(* Logix 5000 project; controller TEC_81 vendor 1 type 14 code 148 rev 36.11; software revision 36.00 *)

TASK MainTask (continuous, watchdog 500 ms) : MainProgram, _05_Mesa_Central, _Almacen_2, _Almacen_1, Manu_camaras, CNC1_Prueba
TASK SafetyTask (periodic, rate 20 ms, priority 10, watchdog 20 ms) : SafetyProgram

MODULES
   Local : vendor 1 type 14 code 148 (ICP 1, rev 36.11)
      Ethernet : vendor 1 type 12 code 200 (ICP 0, Ethernet 10.12.143.10, rev 10.7, Input RPI 500 ms)
           Point_IO_Conveyor_2:4:I.0   // Cambio de Dirección Extendido Lado A Almacén
           Point_IO_Conveyor_2:4:I.1   // Cambio de Dirección Retraido Lado A Almacén
           Point_IO_Conveyor_2:4:I.2   // Sensor Inductivo Lado B CNC (Entrada)
           Point_IO_Conveyor_2:4:I.4   // Spare
           Point_IO_Conveyor_2:4:I.5   // Spare
           Point_IO_Conveyor_2:4:I.3   // Sensor Inductivo Posición Lado B CNC
           Point_IO_Conveyor_2:4:I.7   // Sensor Inductivo Lado A Almacen (Entrada)
           Point_IO_Conveyor_2:4:I.6   // Sensor Inductivo Posición Lado A CNC
           Point_IO_Conveyor_1:10:O.0   // Spare
           Point_IO_Conveyor_1:10:O.1   // Spare
           Point_IO_Conveyor_1:10:O.2   // Spare
           Point_IO_Conveyor_1:10:O.3   // Spare
           Point_IO_Conveyor_1:10:O.4   // Spare
           Point_IO_Conveyor_1:10:O.5   // Spare
           Point_IO_Conveyor_1:10:O.6   // Spare
           Point_IO_Conveyor_1:10:O.7   // Spare
           Point_IO_Conveyor_2:8:O.0   // Spare
           Point_IO_Conveyor_2:8:O.1   // Spare
           Point_IO_Conveyor_2:8:O.2   // Spare
           Point_IO_Conveyor_2:8:O.3   // Spare
           Point_IO_Conveyor_2:8:O.4   // Spare
           Point_IO_Conveyor_2:8:O.5   // Spare
           Point_IO_Conveyor_2:8:O.6   // Spare
           Point_IO_Conveyor_2:8:O.7   // Spare
           MesaCentral:3:O.0   // Bobina Interlock Entrada CNC
           MesaCentral:3:O.1   // Pistón Esquina Extendido Mesa Kuka
           MesaCentral:3:O.3   // Piston Central Extendido Mesa Kuka
           MesaCentral:3:O.2   // Piston Centro Retraido Mesa Kuka
           Point_IO_Conveyor_1:4:I.7   // Sensor Inductivo Lado A Almacen (Entrada)
           Point_IO_Conveyor_1:4:I.2   // Sensor Inductivo Lado CNC (Entrada)
           Point_IO_Conveyor_1:4:I.4   // Spare
           Point_IO_Conveyor_1:4:I.5   // Spare
           Point_IO_Conveyor_1:4:I.0   // Cambio de Dirección Extendido Lado A
           Point_IO_Conveyor_1:4:I.3   // Sensor Inductivo Posición Lado B CNC
           Point_IO_Conveyor_1:4:I.6   // Sensor Inductivo Posición Lado A CNC
           Point_IO_Conveyor_1:4:I.1   // Cambio de Dirección Retraido Lado A
           Point_IO_Conveyor_1:9:O.0   // Spare
           Point_IO_Conveyor_1:9:O.1   // Spare
           Point_IO_Conveyor_1:9:O.2   // Spare
           Point_IO_Conveyor_1:9:O.3   // Spare
           Point_IO_Conveyor_1:9:O.4   // Spare
           Point_IO_Conveyor_1:9:O.5   // Spare
           Point_IO_Conveyor_1:9:O.6   // Spare
           Point_IO_Conveyor_1:9:O.7   // Spare
           MesaCentral:1:I.4   // Sensor Posición Ventosa de Robot Kuka
           MesaCentral:1:I.2   // Sensor Pistón Centro
           MesaCentral:1:I.3   // Sensor Pistón Centro
           MesaCentral:1:I.5   // Sensor Posición Destornillador de Robot Kuka
           MesaCentral:1:I.0   // Sensor Piston Orilla
           MesaCentral:1:I.1   // Sensor Piston Orilla
           MesaCentral:1:I.6   // Sensor Posición Gripper de Robot Kuka
           Point_IO_Conveyor_1:3:I.0   // Spare
           Point_IO_Conveyor_1:3:I.2   // Sensor Piston Tope CNC
           Point_IO_Conveyor_1:3:I.1   // Sensor Tope Piston Horizontal (Salida de conveyor)
           Point_IO_Conveyor_1:3:I.5   // Sensor Piston Tope Camara Vision
           Point_IO_Conveyor_1:3:I.3   // Sensor Piston Tope Marcadora Laser
           Point_IO_Conveyor_1:3:I.6   // Cambio de Dirección Extendido Lado B
           Point_IO_Conveyor_1:3:I.7   // Cambio de Dirección Retraido Lado B
           Point_IO_Conveyor_1:3:I.4   // Límit Switch Arriba
           Point_IO_Conveyor_1:8:O.0   // Spare
           Point_IO_Conveyor_1:8:O.1   // Spare
           Point_IO_Conveyor_1:8:O.2   // Spare
           Point_IO_Conveyor_1:8:O.3   // Spare
           Point_IO_Conveyor_1:8:O.4   // Spare
           Point_IO_Conveyor_1:8:O.5   // Spare
           Point_IO_Conveyor_1:8:O.6   // Spare
           Point_IO_Conveyor_1:8:O.7   // Spare
           Point_IO_Conveyor_2:10:O.0   // Spare
           Point_IO_Conveyor_2:10:O.1   // Spare
           Point_IO_Conveyor_2:10:O.2   // Spare
           Point_IO_Conveyor_2:10:O.3   // Spare
           Point_IO_Conveyor_2:10:O.4   // Spare
           Point_IO_Conveyor_2:10:O.5   // Spare
           Point_IO_Conveyor_2:10:O.6   // Spare
           Point_IO_Conveyor_2:10:O.7   // Spare
           Point_IO_Conveyor_2:3:I.0   // Spare
           Point_IO_Conveyor_2:3:I.1   // Sensor Tope Piston Horizontal (Salida de conveyor)
           Point_IO_Conveyor_2:3:I.2   // Sensor Piston Tope CNC
           Point_IO_Conveyor_2:3:I.6   // Cambio de Dirección Extendido Lado B CNC
           Point_IO_Conveyor_2:3:I.7   // Cambio de Dirección Retraido Lado B CNC
           Point_IO_Conveyor_2:3:I.3   // Sensor Piston Tope Marcadora Laser
           Point_IO_Conveyor_2:3:I.5   // Sensor Piston Tope Camara Vision
           Point_IO_Conveyor_2:3:I.4   // Límit Switch Arriba
           Point_IO_Conveyor_1:5:I.0   // Sensor Limit Switch Tope
           Point_IO_Conveyor_1:5:I.1   // Sensor Limit Inductivo Posición Tope Corredizo (almacen)
           Point_IO_Conveyor_1:5:I.2   // Spare
           Point_IO_Conveyor_1:5:I.3   // Spare
           Point_IO_Conveyor_1:5:I.4   // Spare
           Point_IO_Conveyor_1:5:I.5   // Spare
           Point_IO_Conveyor_1:5:I.6   // Spare
           Point_IO_Conveyor_1:5:I.7   // Spare
           Point_IO_Conveyor_2:5:I.0   // Sensor Limit Switch Tope
           Point_IO_Conveyor_2:5:I.1   // Sensor Inductivo Posición Tope Corredizo (Salida a Almacen)
           Point_IO_Conveyor_2:5:I.2   // Robot Fanuc Fence Open
           Point_IO_Conveyor_2:5:I.4   // Spare
           Point_IO_Conveyor_2:5:I.5   // Spare
           Point_IO_Conveyor_2:5:I.6   // Spare
           Point_IO_Conveyor_2:5:I.7   // Spare
           Point_IO_Conveyor_2:5:I.3   // Robot Fanuc E Stop
           Point_IO_Conveyor_2:1:I.0   // Spare
           Point_IO_Conveyor_2:1:I.1   // Spare
           Point_IO_Conveyor_2:1:I.2   // Botón Negro Puerta
           Point_IO_Conveyor_2:1:I.5   // Spare
           Point_IO_Conveyor_2:1:I.6   // Sensor Difuso Presencia Lado A Almacen 1-1
           Point_IO_Conveyor_2:1:I.7   // Sensor Difuso Presencia Lado A Almacen 1-2
           Point_IO_Conveyor_2:1:I.4   // Contacto Auxiliar Escaner de Seguridad
           Point_IO_Conveyor_2:1:I.3   // Botón Rojo Puerta
           MesaCentral:2:I.1   // Reset Puerta CNC
           MesaCentral:2:I.3   // Emergency Stop Puerta CNC
           MesaCentral:2:I.2   // Enable Puerta CNC
           Point_IO_Conveyor_1:6:I.0   // Spare
           Point_IO_Conveyor_1:6:I.1   // Spare
           Point_IO_Conveyor_1:6:I.2   // Spare
           Point_IO_Conveyor_1:6:I.3   // Spare
           Point_IO_Conveyor_1:6:I.4   // Spare
           Point_IO_Conveyor_1:6:I.5   // Spare
           Point_IO_Conveyor_1:6:I.6   // Spare
           Point_IO_Conveyor_1:6:I.7   // Spare
           Point_IO_Conveyor_2:7:O.3   // Tope Pison Marcadora Laser (Freno 06)
           Point_IO_Conveyor_2:7:O.0   // Piston Horizontal Para Salida de Pieza
           Point_IO_Conveyor_2:7:O.4   // Subir Limit Switch
           Point_IO_Conveyor_2:7:O.1   // Tope Piston Salida de Producto (freno 8)
           Point_IO_Conveyor_2:7:O.2   // Tope Piston CNC (Freno 5)
           Point_IO_Conveyor_2:7:O.5   // Tope Piston Cámara Visión
           Point_IO_Conveyor_2:7:O.7   // Piston Cambio de Dirección Almacén
           Point_IO_Conveyor_2:7:O.6   // Piston Cambio de Dirección CNC
           Point_IO_Conveyor_1:2:I.0   // Sensor difuso presencia lado B Almacen 2-1 (Robot)
           Point_IO_Conveyor_1:2:I.2   // Sensor Difuso Lado A CNC 3-1 (Centro-Marcadora Laser)
           Point_IO_Conveyor_1:2:I.3   // Sensor Difuso Lado A CNC 3-2 (Centro-Marcadora Laser)
           Point_IO_Conveyor_1:2:I.7   // Spare
           Point_IO_Conveyor_1:2:I.4   // Sensor Piston Horizontal Extendido
           Point_IO_Conveyor_1:2:I.5   // Sensor Piston Horizontal Retraido
           Point_IO_Conveyor_1:2:I.1   // Sensor difuso presencia lado B Almacen 2-2 (Robot)
           Point_IO_Conveyor_1:2:I.6   // Sensor Inductivo Presencia en Zona de Vision (Actual Marcadora Laser)
           Point_IO_Conveyor_2:6:I.0   // Spare
           Point_IO_Conveyor_2:6:I.1   // Spare
           Point_IO_Conveyor_2:6:I.2   // Spare
           Point_IO_Conveyor_2:6:I.3   // Spare
           Point_IO_Conveyor_2:6:I.4   // Spare
           Point_IO_Conveyor_2:6:I.5   // Spare
           Point_IO_Conveyor_2:6:I.6   // Spare
           Point_IO_Conveyor_2:6:I.7   // Spare
           Point_IO_Conveyor_2:9:O.0   // Spare
           Point_IO_Conveyor_2:9:O.1   // Spare
           Point_IO_Conveyor_2:9:O.2   // Spare
           Point_IO_Conveyor_2:9:O.3   // Spare
           Point_IO_Conveyor_2:9:O.4   // Spare
           Point_IO_Conveyor_2:9:O.5   // Spare
           Point_IO_Conveyor_2:9:O.6   // Spare
           Point_IO_Conveyor_2:9:O.7   // Spare
           Point_IO_Conveyor_2:2:I.0   // Sensor Difuso Presencia Lado B CNC 2-1
           Point_IO_Conveyor_2:2:I.1   // Sensor Difuso Presencia Lado B CNC 2-2
           Point_IO_Conveyor_2:2:I.2   // Sensor Difuso Presencia Lado A CNC 3-1
           Point_IO_Conveyor_2:2:I.4   // Sensor Inductivo Presente Zona de Marcadora Láser
           Point_IO_Conveyor_2:2:I.5   // Sensor Piston Horizontal Retraido
           Point_IO_Conveyor_2:2:I.7   // Spare
           Point_IO_Conveyor_2:2:I.3   // Sensor Difuso Presencia Lado A CNC 3-2
           Point_IO_Conveyor_2:2:I.6   // Sensor Piston Horizontal Extendido
           Point_IO_Conveyor_1:7:O.3   // Tope Pison Marcadora Laser (Freno 06)
           Point_IO_Conveyor_1:7:O.5   // Tope Piston Cámara Visión
           Point_IO_Conveyor_1:7:O.2   // Tope Piston CNC (Freno 5)
           Point_IO_Conveyor_1:7:O.1   // Tope Piston Salida de Producto (Freno 8)
           Point_IO_Conveyor_1:7:O.0   // Piston Horizontal Para Salida de Pieza
           Point_IO_Conveyor_1:7:O.6   // Piston Cambio de Dirección CNC
           Point_IO_Conveyor_1:7:O.7   // Piston Cambio de Dirección Almacén
           Point_IO_Conveyor_1:7:O.4   // Subir Limit Switch
           Point_IO_Conveyor_1:1:I.0   // Spare
           Point_IO_Conveyor_1:1:I.1   // Spare
           Point_IO_Conveyor_1:1:I.5   // Spare
           Point_IO_Conveyor_1:1:I.6   // Sensor difuso presencia lado A Almacen 1-1
           Point_IO_Conveyor_1:1:I.7   // Sensor difuso presencia lado A Almacen 1-2
           Point_IO_Conveyor_1:1:I.4   // Auxiliar Scanner de Seguridad (Sin Conexión)
           Point_IO_Conveyor_1:1:I.2   // Boton negro Puerta
           Point_IO_Conveyor_1:1:I.3   // Boton Rojo Puerta
         Almacen2 : vendor 1 type 37 code 48 (Ethernet 10.12.143.9, rev 7.1, MotionDiagnostics RPI 1 ms, MotionSync RPI 2 ms)
         Almacen_1 : vendor 1 type 37 code 48 (Ethernet 10.12.143.8, rev 7.1, MotionDiagnostics RPI 1 ms, MotionSync RPI 2 ms)
         Fanuc_M10iA : vendor 356 type 12 code 2 (Ethernet 10.12.143.28, rev 2.4, StandardDataDriven RPI 32 ms)
         Fanuc_Delta : vendor 356 type 12 code 2 (Ethernet 10.12.143.47, rev 2.2, StandardDataDriven RPI 32 ms)
              Fanuc_Delta:I1.Input[0].0   // cmd enabled
              Fanuc_Delta:I1.Input[0].2   // prg running
              Fanuc_Delta:I1.Input[0].4   // motion held
              Fanuc_Delta:I1.Input[0].6   // at perch
              Fanuc_Delta:I1.Input[2].3   // reserved
              Fanuc_Delta:I1.Input[0].1   // system ready
              Fanuc_Delta:I1.Input[0].3   // prg paused
              Fanuc_Delta:I1.Input[1].1   // busy
              Fanuc_Delta:I1.Input[1].2   // ack1
              Fanuc_Delta:I1.Input[0].7   // tp enabled
              Fanuc_Delta:I1.Input[0].5   // fault
              Fanuc_Delta:I1.Input[1].3   // ack2
              Fanuc_Delta:I1.Input[2].2   // snack
              Fanuc_Delta:I1.Input[1].0   // batt alarm
              Fanuc_Delta:I1.Input[1].4   // ack3
              Fanuc_Delta:I1.Input[1].5   // ack4
              Fanuc_Delta:I1.Input[1].6   // ack5
              Fanuc_Delta:I1.Input[1].7   // ack6
              Fanuc_Delta:I1.Input[2].0   // ack7
              Fanuc_Delta:I1.Input[2].1   // ack8
              Fanuc_Delta:O1.Output[0].4   // fault reset
              Fanuc_Delta:O1.Output[0].0   // IMSTP
              Fanuc_Delta:O1.Output[0].2   // SFSPD
              Fanuc_Delta:O1.Output[0].3   // cycle stop
              Fanuc_Delta:O1.Output[2].0   // pns strobe
              Fanuc_Delta:O1.Output[0].7   // Enable
              Fanuc_Delta:O1.Output[2].1   // prod start
              Fanuc_Delta:O1.Output[0].1   // hold
              Fanuc_Delta:O1.Output[0].6   // Home
              Fanuc_Delta:O1.Output[1].0   // rsr1
              Fanuc_Delta:O1.Output[1].1   // rsr2
              Fanuc_Delta:O1.Output[0].5   // start
              Fanuc_Delta:O1.Output[1].2   // rsr3
              Fanuc_Delta:O1.Output[1].3   // rsr4
              Fanuc_Delta:O1.Output[1].4   // rsr5
              Fanuc_Delta:O1.Output[1].5   // rsr6
              Fanuc_Delta:O1.Output[1].6   // rsr7
              Fanuc_Delta:O1.Output[1].7   // rsr8
              Fanuc_Delta:O1.Output[2].5   // 22
              Fanuc_Delta:O1.Output[2].6   // 23
         Point_IO_Conveyor_2 : 1734-AENTR (Ethernet 10.12.143.43, rev 5.12, Output RPI 20 ms)   // Lado Izquierdo
            E01N023S03 : 1734-IB8 (PointIO 3, rev 3.22)
            E01N023S06 : 1734-IB8 (PointIO 6, rev 3.22)
            E01N023S05 : 1734-IB8 (PointIO 5, rev 3.22)
            E01N023S04 : 1734-IB8 (PointIO 4, rev 3.22)
            E01N023S01 : 1734-IB8 (PointIO 1, rev 3.22)
            E01N023S02 : 1734-IB8 (PointIO 2, rev 3.22)
            E01N023S0 : 1734-OB8 (PointIO 7, rev 3.22)
            E01N023S08 : 1734-OB8 (PointIO 8, rev 3.22)
            E01N023S10 : 1734-OW4 (PointIO 10, rev 3.22)
            E01N023S09 : 1734-OW4 (PointIO 9, rev 3.22)
            E01N023S12 : vendor 1 type 35 code 16 (PointIO 12, rev 2.2, Input RPI 10 ms, Output RPI 20 ms)
                 Point_IO_Conveyor_2:12:O.Pt01Data   // S2 PowerFlex Transportador 2
                 Point_IO_Conveyor_2:12:O.Pt07Data   // Spare
                 Point_IO_Conveyor_2:12:O.Pt06Data   // Spare
                 Point_IO_Conveyor_2:12:O.Pt00Data   // S1 PowerFlex Transportador 2
                 Point_IO_Conveyor_2:12:O.Pt04Data   // S1 Robot External E Stop Relay 2
                 Point_IO_Conveyor_2:12:O.Pt03Data   // S2 Robot External E-stop Relay 1
                 Point_IO_Conveyor_2:12:O.Pt02Data   // S1 Robot External E-stop Relay 1
                 Point_IO_Conveyor_2:12:O.Pt05Data   // S2 Robot External E Stop Relay 2
            E01N023S11 : vendor 1 type 35 code 15 (PointIO 11, rev 2.2, Input RPI 10 ms, Output RPI 20 ms)
                 Point_IO_Conveyor_2:11:I.Pt07Data   // Spare
                 Point_IO_Conveyor_2:11:I.Pt01Data   // Spare
                 Point_IO_Conveyor_2:11:I.Pt05Data   // Scanner
                 Point_IO_Conveyor_2:11:I.Pt02Data   // E_Stop Coneyor 2 Lierado
                 Point_IO_Conveyor_2:11:I.Pt06Data   // Spare
                 Point_IO_Conveyor_2:11:I.Pt00Data   // Spare
                 Point_IO_Conveyor_2:11:I.Pt04Data   // Scanner
                 Point_IO_Conveyor_2:11:I.Pt03Data   // E_Stop Coneyor 2 Presionado
         Point_IO_Conveyor_1 : 1734-AENTR (Ethernet 10.12.143.42, rev 5.12, Output RPI 20 ms)
            E01N022S04 : 1734-IB8 (PointIO 4, rev 3.22)
            E01N022S03 : 1734-IB8 (PointIO 3, rev 3.22)
            E01N022S02 : 1734-IB8 (PointIO 2, rev 3.22)
            E01N022S06 : 1734-IB8 (PointIO 6, rev 3.22)
            E01N022S05 : 1734-IB8 (PointIO 5, rev 3.22)
            E01N022S01 : 1734-IB8 (PointIO 1, rev 3.22)
            E01N022S07 : 1734-OB8 (PointIO 7, rev 3.22)
            E01N022S08 : 1734-OB8 (PointIO 8, rev 3.22)
            E01N022S09 : 1734-OW4 (PointIO 9, rev 3.22)
            E01N022S10 : 1734-OW4 (PointIO 10, rev 3.22)
            E01N022S12 : vendor 1 type 35 code 16 (PointIO 12, rev 2.2, Input RPI 10 ms, Output RPI 20 ms)
                 Point_IO_Conveyor_1:12:O.Pt04Data   // Spare
                 Point_IO_Conveyor_1:12:O.Pt01Data   // S2 PowerFlex Transportador 1
                 Point_IO_Conveyor_1:12:O.Pt03Data   // Spare
                 Point_IO_Conveyor_1:12:O.Pt02Data   // Spare
                 Point_IO_Conveyor_1:12:O.Pt07Data   // Spare
                 Point_IO_Conveyor_1:12:O.Pt05Data   // Spare
                 Point_IO_Conveyor_1:12:O.Pt06Data   // Spare
                 Point_IO_Conveyor_1:12:O.Pt00Data   // S1 PowerFlex Transportador 1
            E01N022S011 : vendor 1 type 35 code 15 (PointIO 11, rev 2.2, Output RPI 20 ms, Input RPI 10 ms)
                 Point_IO_Conveyor_1:11:I.Pt07Data   // Spare
                 Point_IO_Conveyor_1:11:I.Pt02Data   // Spare
                 Point_IO_Conveyor_1:11:I.Pt00Data   // E_Stop Conveyor 1 Liberado
                 Point_IO_Conveyor_1:11:I.Pt05Data   // Spare
                 Point_IO_Conveyor_1:11:I.Pt06Data   // Spare
                 Point_IO_Conveyor_1:11:I.Pt04Data   // Spare
                 Point_IO_Conveyor_1:11:I.Pt03Data   // Spare
                 Point_IO_Conveyor_1:11:I.Pt01Data   // E_Stop Conveyor 1 Presionado
         Point_IO_Almacen_2 : 1734-AENTR (Ethernet 10.12.143.41, rev 5.12, Output RPI 20 ms)   // Almacen Lado Derecho
            E01020S02 : 1734-IB8 (PointIO 2, rev 3.22)
            E01N021S07 : vendor 1 type 35 code 16 (PointIO 7, rev 2.2, Output RPI 20 ms, Input RPI 10 ms)
            E01N021S06 : vendor 1 type 35 code 15 (PointIO 6, rev 2.2, Input RPI 10 ms, Output RPI 20 ms)
         Point_IO_Almacen1 : 1734-AENTR (Ethernet 10.12.143.40, rev 5.12, Output RPI 20 ms)
            Point_IO_Almacen1_2 : 1734-IB8 (PointIO 2, rev 3.22)
            E01020S06 : vendor 1 type 35 code 15 (PointIO 6, rev 2.2, Output RPI 20 ms, Input RPI 10 ms)
            E01020S07 : vendor 1 type 35 code 16 (PointIO 7, rev 2.2, Input RPI 10 ms, Output RPI 20 ms)
                 Point_IO_Almacen1:7:O.Pt02Data   // Interlock 2 Release Coil
         MesaCentral : 1734-AENTR (Ethernet 10.12.143.46, rev 5.11, Output RPI 20 ms)
            EN01N030S02 : 1734-IB8 (PointIO 2, rev 3.22)
            EN01N030S01 : 1734-IB8 (PointIO 1, rev 3.22)
            EN01N030S03 : 1734-OW4 (PointIO 3, rev 3.22)
            OB8S_MesaKuka : vendor 1 type 35 code 16 (PointIO 5, rev 2.2, Input RPI 10 ms, Output RPI 20 ms)
                 MesaCentral:5:O.Pt00Data   // Interlock 1 Release Coil
            EN01N030S04 : vendor 1 type 35 code 15 (PointIO 4, rev 2.2, Input RPI 10 ms, Output RPI 20 ms)
                 MesaCentral:4:I.Pt02Data   // Interlock paro de emergenia
                 MesaCentral:4:I.Pt01Data   // Contacto 2 puerta de entrada cnc
                 MesaCentral:4:I.Pt00Data   // Contacto 1 puerta de entrada cnc
                 MesaCentral:4:I.Pt03Data   // Interlock paro de emergenia contacto 2
         Almacen_2 : vendor 1 type 14 code 235 (Ethernet 10.12.143.18, rev 31.12, $3a1ccfee$ RPI 20 ms, $23a22c79$ RPI 20 ms, $37d2c9b8$ RPI 20 ms, $dae8255b$ RPI 20 ms, $f8b61452$ RPI 20 ms, $1288edcd$ RPI 20 ms, $c7c1ea3c$ RPI 20 ms, $5129664f$ RPI 20 ms, $9b9df9f6$ RPI 20 ms, $af419361$ RPI 20 ms)
         Almacen1 : vendor 1 type 14 code 235 (Ethernet 10.12.143.17, rev 33.11, $f6b484da$ RPI 20 ms, $7a7e9135$ RPI 20 ms, $47cb4104$ RPI 20 ms, $eccb3ef7$ RPI 20 ms, $156cf8fe$ RPI 20 ms, $8b409b49$ RPI 20 ms, $dfe4ff48$ RPI 20 ms)
         CNC_1 : 1791ES-IB8XOBV4 (Ethernet 10.12.143.44, rev 1.9, Input RPI 10 ms, Output RPI 20 ms)
              CNC_1:I.Pt01Data   // Door Closed Sensor
              CNC_1:O.Pt00Data   // S1 CNC 1 E Stop
              CNC_1:O.Pt02Data   // Close Door Piston CNC 1
         CNC_2 : 1791ES-IB8XOBV4 (Ethernet 10.12.143.45, rev 1.9, Output RPI 20 ms, Input RPI 10 ms)
              CNC_2:O.Pt03Data   // S2 CNC 2 E Stop
              CNC_2:O.Pt00Data   // S1 CNC 2 E Stop
      @fcc730f7@:Partner : vendor 1 type 14 code 146 (ICP 2, rev 36.11)
END_MODULES

VAR_GLOBAL   (* controller tags *)
   Abrir_Prensa_CNC_1 : BOOL;   // Señal Para Abrir Prensa en CNC 1
   Abrir_Prensa_CNC_1_Safety : BOOL;   // Abrir Prensa CNC 1
   Abrir_Prensa_CNC_2 : BOOL;   // START CYCLE CNC 2
   Abrir_Prensa_CNC_2_Safety : BOOL;
   AbrirInterlock_conveyor_Control : BOOL;
   AbrirInterlock_conveyor_Safety : BOOL;   // Mapped green button for interlock 2 opening
   AbrirInterlock_Principal_Control : BOOL;
   AbrirInterlock_Principal_Safety : BOOL;   // Mapped green button for interlock 1 opening
   Alm2_GripperClosed : BOOL;
   Alm2_GripperOpen : BOOL;
   Alm2_Home : BOOL;
   Alm2_S1 : BOOL;   // Turn to Storage
   Alm2_S2 : BOOL;   // Turn to Conveyor
   Alm2_X1 : BOOL;   // Storage Left
   Alm2_X2 : BOOL;   // Storage Rigth
   Alm2_Z1 : BOOL;   // Side Conveyor
   Alm2_Z2 : BOOL;   // Side Storage
   AlmPosReq : DINT;
   Alw_OFF : BOOL; {constant}
   Auto_Conv_1 : BOOL := 1;   // Secuencia Activada Automática Conveyor 1
   Axis2_Home : MOTION_INSTRUCTION;
   Axis_1 : AXIS_CIP_DRIVE;
   Axis_2 : AXIS_CIP_DRIVE;   // Almacen 2
   B_Reset_Posicion_kinetix : DINT := 319;
   B_Reset_Posicion_kinetix_1 : DINT;
   Btn_Negro_Conv_1 : BOOL;   // Botón Negro Puerta de Conveyor 1
   Btn_Negro_Conv_2 : BOOL;   // Botón Negro Puerta de Conveyor 2
   Btn_Rojo_Conv_1 : BOOL;   // Botón Rojo Puerta de Conveyor 1
   Btn_Rojo_Conv_2 : BOOL;   // Botón Rojo Puerta de Conveyor 2
   CambioDir_Ext_Almacen_Conv_1 : BOOL;   // Sensor Cambio de Dirección Extendido Lado A (Almacén)
   CambioDir_Ext_Almacen_Conv_2 : BOOL;   // Sensor Cambio de Dirección Extendido Lado A Almacén
   CambioDir_Ext_CNC_Conv_1 : BOOL;   // Sensor Cambio de Dirección Extendido Lado B (CNC)
   CambioDir_Ext_CNC_Conv_2 : BOOL;   // Cambio de Dirección Extendido Lado B CNC
   CambioDir_Ret_Almacen_Conv_1 : BOOL := 1;   // Sensor Cambio de Dirección Retraido Lado A (Almacén)
   CambioDir_Ret_Almacen_Conv_2 : BOOL;   // Sensor Cambio de Dirección Retraido Lado A Almacén
   CambioDir_Ret_CNC_Conv_1 : BOOL := 1;   // Sensor Cambio de Dirección Retraido Lado B (CNC)
   CambioDir_Ret_CNC_Conv_2 : BOOL;   // Cambio de Dirección Retraido Lado B CNC
   Cerrar_Prensa_CNC_1 : BOOL;   // Señal Para Cerrar Prensa en CNC 1
   Cerrar_Prensa_CNC_1_Safety : BOOL;   // Cerrar Prensa CNC 1
   Cerrar_Prensa_CNC_2 : BOOL;   // Señal Para Cerrar Prensa en CNC 2
   Cerrar_Prensa_CNC_2_Safety : BOOL;
   Cfg_Pos_Test : BOOL := 1;
   Close_Door_CNC_1_Control : BOOL;   // Cerrar Puerta CNC 1 Secuencia de Control Fanuc Fuera de CNC 1
   Close_Door_CNC_1_Safety : BOOL;   // Cerrar Puerta de CNC 1 Desde ArmorBlock
   Close_Door_CNC_2_Control : BOOL;   // Cerrar Puerta CNC 2 Secuencia de Control Fanuc Fuera de CNC 2
   Close_Door_CNC_2_Safety : BOOL;   // Cerrar Puerta de CNC 2 Desde ArmorBlock
   Close_Griper_Fanuc : BOOL;   // Señal de Griper Cerrado Robot Fanuc
   Cmd_Axis_2 : BOOL;
   Cmd_OnDly : TIMER;
   Cmd_Pos : DINT := 380;
   Cmd_Robot_Conv_1 : BOOL;
   Cmd_Robot_Conv_2 : BOOL := 1;
   Cmd_YPickSafe : BOOL;
   Cmd_YPickSafe_Alm1 : BOOL;
   Cmd_YPlaceSafe : BOOL;
   Cmd_YPlaceSafe_Alm1 : BOOL;
   Cmd_YSafePos : BOOL;
   Cmd_YSafePos_Alm1 : BOOL;
   Cmd_YtoYOff : BOOL;
   Cmd_YtoYOff_Alm1 : BOOL;
   Cmd_YtoYPick : BOOL;
   Cmd_YtoYPick_Alm1 : BOOL;
   Cmd_YtoYPlace : BOOL;
   Cmd_YtoYPlace_Alm1 : BOOL;
   Cmd_YtoYPlaceOffset : BOOL;
   Cmd_YtoYPlaceOffset_Alm1 : BOOL;
   CNC_1_Cerrar_Prensa : BOOL;   // Señal de salida para Cerrar prensa en CNC 1
   CNC_1_Confirma_Terminado_Pieza : BOOL := 1;   // Señal del CNC 1 de Pieza Terminada
   CNC_1_Wrk : BOOL;
   CNC_2_Confirma_Terminado_Pieza : BOOL;   // Señal del CNC 2 de Pieza Terminada
   CNC_2_Wrk : BOOL := 1;
   com_ok_PLC : Safety; {produced, access Read Only}
   Consumeded_Signals_Conveyor_1_TEC_81 : DINT := 256;
   Conv_1_Vacio_Inicial : BOOL := 1;   // Bit de Verificación Conveyor 1 Vacio
   Conveyor_1_Tomar_Pieza : BOOL;   // Señal del Conveyor 1 para Tomar Pieza Iniciar Ciclo
   Conveyor_2_Tomar_Pieza : BOOL;   // Señal del Conveyor 2 para Tomar Pieza Iniciar Ciclo
   Ctrl_Kinetix_A2 : DINT := 1;   // Boton Start Kinetix
   CycleStartDly : TIMER;
   Destino_Fanuc_Cerrar_Griper : BOOL := 1;   // Salida de Aviso al Robot Fanuc de Cerrar Griper
   Destino_Fanuc_Confirmar_Pieza_Libre : BOOL;   // Salida de Aviso al Robot Fanuc Pieza libre para ser tomada
   Destino_Fanuc_Confirmar_Pieza_Presionada : BOOL;
   Destino_Fanuc_Pick_Conveyor_1 : BOOL;
   Destino_Fanuc_Pick_Conveyor_2 : BOOL;
   Destino_Fanuc_Place_CNC_1 : BOOL;
   Destino_Fanuc_Place_CNC_2 : BOOL;
   Destino_Fanuc_Place_Mesa_Kuka_1 : BOOL;
   Destino_Fanuc_Place_Mesa_Kuka_2 : BOOL;
   Destino_Fanuc_Posicion_Segura_Conveyor_1 : BOOL;
   Destino_Fanuc_Wait : BOOL;
   Destino_Pick_CNC_1 : BOOL;
   Destino_Pick_CNC_2 : BOOL;
   Destino_Pick_Conveyor_2 : BOOL := 1;
   Destino_Pick_Mesa_Kuka_1 : BOOL;
   Destino_Pick_Mesa_Kuka_2 : BOOL;
   Destino_Place_Conveyor_1 : BOOL;
   Destino_Place_Conveyor_2 : BOOL;
   DestornilladorEnPosicion_Mesa : BOOL;   // Sensor de posición de Destornillador en Mesa Central
   Dly : TIMER[16];
   Done_Kinetx : DINT; {produced}
   Done_Kinetx_1 : DINT;
   Done_Step_00_Robot : BOOL;
   Done_Step_10_Robot : BOOL;
   Done_Step_11_Robot : BOOL;
   Done_Step_12_Robot : BOOL;
   Done_Step_13_Robot : BOOL;
   Done_Step_14_Robot : BOOL;
   Done_Step_15_Robot : BOOL;
   Done_Step_16_Robot : BOOL;
   Done_Step_17_Robot : BOOL;
   Done_Step_18_Robot : BOOL;
   Done_Step_19_Robot : BOOL;
   Done_Step_200_Pieza : BOOL;
   Done_Step_200A_Pieza : BOOL;
   Done_Step_201_Pieza : BOOL;
   Done_Step_201A_Pieza : BOOL;
   Done_Step_202_Pieza : BOOL;
   Done_Step_203_Pieza : BOOL;
   Done_Step_204_Pieza : BOOL;
   Done_Step_205_Pieza : BOOL;
   Done_Step_206_Pieza : BOOL;
   Done_Step_207_Pieza : BOOL;
   Done_Step_208_Pieza : BOOL;
   Done_Step_209_Pieza : BOOL;
   Done_Step_209A_Pieza : BOOL;
   Done_Step_20_Robot : BOOL;
   Done_Step_210_Pieza : BOOL;
   Done_Step_211_Pieza : BOOL;
   Done_Step_212_Pieza : BOOL;
   Done_Step_213_Pieza : BOOL;
   Done_Step_214_Pieza : BOOL;
   Done_Step_215_Pieza : BOOL;
   Done_Step_216_Pieza : BOOL;
   Done_Step_217_Pieza : BOOL;
   Done_Step_217A_Pieza : BOOL;
   Done_Step_218_Pieza : BOOL;
   Done_Step_219_Pieza : BOOL;
   Done_Step_21_Robot : BOOL;
   Done_Step_220_Pieza : BOOL;
   Done_Step_221_Pieza : BOOL;
   Done_Step_221A_Pieza : BOOL;
   Done_Step_222_Pieza : BOOL;
   Done_Step_223_Pieza : BOOL;
   Done_Step_224_Pieza : BOOL;
   Done_Step_225_Pieza : BOOL;
   Done_Step_226_Pieza : BOOL;
   Done_Step_227_Pieza : BOOL;
   Done_Step_228_Pieza : BOOL;
   Done_Step_229_Pieza : BOOL;
   Done_Step_22_Robot : BOOL;
   Done_Step_230_Pieza : BOOL;
   Done_Step_231_Pieza : BOOL;
   Done_Step_232_Pieza : BOOL;
   Done_Step_233_Pieza : BOOL;
   Done_Step_234_Pieza : BOOL;
   Done_Step_235_Pieza : BOOL;
   Done_Step_236_Pieza : BOOL;
   Done_Step_237_Pieza : BOOL;
   Done_Step_238_Pieza : BOOL;
   Done_Step_239_Pieza : BOOL;
   Done_Step_23_Robot : BOOL;
   Done_Step_240_Pieza : BOOL;
   Done_Step_241_Pieza : BOOL;
   Done_Step_24_Robot : BOOL;
   Done_Step_25_Robot : BOOL;
   Done_Step_26_Robot : BOOL;
   Done_Step_300_Pieza_2 : BOOL;
   Done_Step_301_Pieza_2 : BOOL;
   Done_Step_302_Pieza_2 : BOOL;
   Done_Step_303_Pieza_2 : BOOL;
   Done_Step_304_Pieza_2 : BOOL;
   Done_Step_304A_Pieza_2 : BOOL;
   Done_Step_304B_Pieza_2 : BOOL;
   Done_Step_305_Pieza_2 : BOOL;
   Done_Step_306_Pieza_2 : BOOL;
   Done_Step_307_Pieza_2 : BOOL;
   Done_Step_308_Pieza_2 : BOOL;
   Done_Step_309_Pieza_2 : BOOL;
   Done_Step_30_Robot : BOOL;
   Done_Step_310_Pieza_2 : BOOL;
   Done_Step_311_Pieza_2 : BOOL;
   Done_Step_312_Pieza_2 : BOOL;
   Done_Step_313_Pieza_2 : BOOL;
   Done_Step_314_Pieza_2 : BOOL;
   Done_Step_315_Pieza_2 : BOOL;
   Done_Step_316_Pieza_2 : BOOL;
   Done_Step_317_Pieza_2 : BOOL;
   Done_Step_318_Pieza_2 : BOOL;
   Done_Step_319_Pieza_2 : BOOL;
   Done_Step_31_Robot : BOOL;
   Done_Step_320_Pieza_2 : BOOL;
   Done_Step_320A_Pieza_2 : BOOL;
   Done_Step_321_Pieza_2 : BOOL;
   Done_Step_322_Pieza_2 : BOOL;
   Done_Step_323_Pieza_2 : BOOL;
   Done_Step_324_Pieza_2 : BOOL;
   Done_Step_325_Pieza_2 : BOOL;
   Done_Step_326_Pieza_2 : BOOL;
   Done_Step_327_Pieza_2 : BOOL;
   Done_Step_328_Pieza_2 : BOOL;
   Done_Step_329_Pieza_2 : BOOL;
   Done_Step_32_Robot : BOOL;
   Done_Step_330_Pieza_2 : BOOL;
   Done_Step_331_Pieza_2 : BOOL;
   Done_Step_332_Pieza_2 : BOOL;
   Done_Step_333_Pieza_2 : BOOL;
   Done_Step_334_Pieza_2 : BOOL;
   Done_Step_335_Pieza_2 : BOOL;
   Done_Step_336_Pieza_2 : BOOL;
   Done_Step_337_Pieza_2 : BOOL;
   Done_Step_338_Pieza_2 : BOOL;
   Done_Step_339_Pieza_2 : BOOL;
   Done_Step_33_Robot : BOOL;
   Done_Step_340_Pieza_2 : BOOL;
   Done_Step_341_Pieza_2 : BOOL;
   Done_Step_342_Pieza_2 : BOOL;
   Done_Step_343_Pieza_2 : BOOL;
   Done_Step_344_Pieza_2 : BOOL;
   Done_Step_345_Pieza_2 : BOOL;
   Done_Step_346_Pieza_2 : BOOL;
   Done_Step_347_Pieza_2 : BOOL;
   Done_Step_348_Pieza_2 : BOOL;
   Done_Step_349_Pieza_2 : BOOL;
   Done_Step_34_Robot : BOOL;
   Done_Step_350_Pieza_2 : BOOL;
   Done_Step_351_Pieza_2 : BOOL;
   Done_Step_352_Pieza_2 : BOOL;
   Done_Step_353_Pieza_2 : BOOL;
   Done_Step_354_Pieza_2 : BOOL;
   Done_Step_355_Pieza_2 : BOOL;
   Done_Step_356_Pieza_2 : BOOL;
   Done_Step_357_Pieza_2 : BOOL;
   Done_Step_358_Pieza_2 : BOOL;
   Done_Step_359_Pieza_2 : BOOL;
   Done_Step_360_Pieza_2 : BOOL;
   Done_Step_40_Robot : BOOL;
   Done_Step_41_Robot : BOOL;
   Done_Step_42_Robot : BOOL;
   Done_Step_43_Robot : BOOL;
   Done_Step_44_Robot : BOOL;
   Done_Step_45_Robot : BOOL;
   Done_Step_46_Robot : BOOL;
   Done_Step_47_Robot : BOOL;
   Done_Step_48_Robot : BOOL;
   Done_Step_50_Robot : BOOL;
   Done_Step_51_Robot : BOOL;
   Done_Step_52_Robot : BOOL;
   Done_Step_53_Robot : BOOL;
   Done_Step_54_Robot : BOOL;
   Done_Step_55_Robot : BOOL;
   Done_Step_56_Robot : BOOL;
   Done_Step_57_Robot : BOOL;
   Done_Step_58_Robot : BOOL;
   EStops_OK : BOOL;   // E-Stop Close Loop Indicator
   EStops_OK_External : DINT := 2; {produced}
   Extender_Piston_1_Mesa_Kuka : BOOL;   // Extender Pistón Esquina de Mesa Central
   Extender_Piston_2_Mesa_Kuka : BOOL;   // Extender Pistón Centro de Mesa Central
   Fanuc_Confirma_Dejar_Pieza : BOOL;   // Confirmación del Robot Fanuc para dejar la pieza
   Fanuc_Confirma_Posicion_Segura : BOOL;   // Posición inical del robot en Cero
   Fanuc_Confirma_Retraido : BOOL;   // Señal de Fanuc en posición segura en Mesa Kuka
   Fanuc_Confirma_Segura_CNC_1 : BOOL;   // Señal del Robot Fanuc para posición Segura en CNC 1
   Fanuc_Confirma_Segura_Conveyor_1 : BOOL;   // Señal Fanuc Posición Segura Conveyor 1
   Fanuc_Confirma_Tomar_Pieza : BOOL;   // Señal de Fanuc en posición para Tomar pieza
   Fanuc_Confirma_TomarDejar_Conveyor_1 : BOOL;   // Señal del Robot Fanuc Posición de Tomar/Dejar en Conveyor 1
   Fanuc_Confirma_TomarDejar_Mesa_1 : BOOL;   // Señal del Robot Fanuc En Posición de dejar Pieza en Pistón 1 Mesa Kuka
   Faul_Axis : DINT;
   From_alm_1 : DINT;
   From_Robot : FromRobot_v02;
        .DO44   // Robot fuera de CNC 2
        .DO62   // ROBOT PLACE
   From_Wh2 : DINT := 4;
   From_Wh2_X : DINT;
   From_Wh2_Y : DINT := 380;
   FromStorage1 : DINT;
   FromStorage1_HomeSeq : DINT;
   FromStorage1_MainSeq : DINT;
   FromStorage_HomeSeq : DINT;   // Alm2
   FromStorage_MainSeq : DINT := 130;   // Alm 2
   GripperEnPosicion_Mesa : BOOL;   // Sensor de posición de Gripper en Mesa Central
   HMI_Fanuc_Mover_A_Mesa_Kuka : BOOL := 1;   // Señal Para el Robot On = Pasar a Mesa Kuka Off = Mover a Dejar a Conveyor
   HMI_Reset_Secuencia : BOOL;
   HMI_Select_Secuencia : BOOL;
   HMI_Start : BOOL;
   home : MOTION_INSTRUCTION;
   Home_Sensor : BOOL;
   In_Pos_Alm_1 : DINT; {produced}
   In_Pos_Alm_2 : DINT; {produced}
   InicioCiclo : BOOL;   // Cycle Start from HMI
   Input_Reset_Almacen_1 : BOOL;
   Input_Reset_almacen_2 : BOOL;
   Input_Reset_Principal : BOOL;
   Input_Reset_Salida_1 : BOOL;
   Int_Robot : INT := 2;
   Int_Robot_2 : INT;
   Int_Robot_ToRobot : ToRobot;
   Interlocks_Ok : BOOL := 1;   // Interlocks Close Loop Indicator
   jaja : BOOL;
   Kinetix_Pos : DINT;
   Kinetix_Pos_Alm_1 : DINT := 64;
   Kinetix_Pos_Alm_2 : DINT := 128;
   KUKA : TIMER;
   KUKA_Posicion_Segura : BOOL;   // Señal de Robot Kuka para indicar que se encuentra en posición segura
   KUKA_Proceso_Terminado_Pieza_1 : BOOL;   // Señal Para Asegurarse de que el Kua Terminó la Pieza 1
   KUKA_Proceso_Terminado_Pieza_2 : BOOL := 1;   // Señal Para Asegurarse de que el Kua Terminó la Pieza 2
   Kuka_Rdy : BOOL;
   Kuka_Termina_Piezas : BOOL;   // Robot Kuka Termina Acabado de Piezas CNC 1 y CNC 2
   Kuka_WrkDn : BOOL;
   LigthCurtain_ok : BOOL;   // Light Curtains Close Loop Indicator
   Limit_UP_Conv_1 : BOOL;   // Subir Limit Switch Conveyor 1
   Limit_UP_Conv_2 : BOOL;   // Subir Limit Switch Conveyor 2
   MAFR_Mtr_Alm_1 : MOTION_INSTRUCTION;
   MAFR_Mtr_Alm_2 : MOTION_INSTRUCTION;
   MainSeq : DINT;
   MAJ_Axis_2 : MOTION_INSTRUCTION; {produced}   // Posicion 5
   MAJ_Axis_2_Dwn : MOTION_INSTRUCTION;
   MAJ_Dir : DINT := 1;
   MAM_1_Mtr_Alm_0 : MOTION_INSTRUCTION;
   MAM_1_Mtr_Alm_1 : MOTION_INSTRUCTION;
   MAM_1_Mtr_Alm_2 : MOTION_INSTRUCTION;
   MAM_2_Mtr_Alm_1 : MOTION_INSTRUCTION;
   MAM_2_Mtr_Alm_2 : MOTION_INSTRUCTION;
   MAM_3_Mtr_Alm_1 : MOTION_INSTRUCTION;
   MAM_3_Mtr_Alm_2 : MOTION_INSTRUCTION;
   MAM_4_Mtr_Alm_1 : MOTION_INSTRUCTION;
   MAM_4_Mtr_Alm_2 : MOTION_INSTRUCTION;
   MAM_5_Mtr_Alm_1 : MOTION_INSTRUCTION;
   MAM_5_Mtr_Alm_2 : MOTION_INSTRUCTION;
   MAM_6_Mtr_Alm_1 : MOTION_INSTRUCTION;
   MAM_6_Mtr_Alm_2 : MOTION_INSTRUCTION;
   MAM_7_Mtr_Alm_2 : MOTION_INSTRUCTION;
   MAM_8_Mtr_Alm_1 : MOTION_INSTRUCTION;
   MAM_8_Mtr_Alm_2 : MOTION_INSTRUCTION;
   MAM_Cmd : MOTION_INSTRUCTION;
   Manual_Conv_1 : BOOL;   // Secuencia Activada Manual Conveyor 1
   MAS_Axis_2 : MOTION_INSTRUCTION;
   MAS_Mtr_Alm_1 : MOTION_INSTRUCTION;
   MAS_Mtr_Alm_2 : MOTION_INSTRUCTION;
   Mayor_Prioridad_Pza_1 : BOOL := 1;   // Bit paraDar Prioridad a la Pieza 1
   Mayor_Prioridad_Pza_2 : BOOL;   // Bit Para Dar prioridad a la pieza 2
   MC : DCI_STOP;
   MC_1_EStop : DCI_STOP;   // Status of E-Stop 1
   MC_1_EStop_Status : BOOL := 1;   // General status of inputs
   MC_1_Interlock : DCI_STOP;   // Status of Interlock 1
   MC_1_Interlock_Status : BOOL := 1;   // General status of inputs
   MC_1_LigthCurtain : DCI_STOP;   // Status of Light Curtain 1
   MC_1_LigthCurtain_Status : BOOL := 1;   // General status of inputs
   MC_2_EStop : DCI_STOP;   // Status of E-Stop 2
   MC_2_EStop_Status : BOOL := 1;   // General status of inputs
   MC_2_Interlock : DCI_STOP;   // Status of Interlock 2
   MC_2_Interlock_Status : BOOL := 1;   // General status of inputs
   MC_2_LightCurtain_Status : BOOL := 1;   // General status of inputs
   MC_2_LigthCurtain : DCI_STOP;   // Status of Light Curtain 2
   MC_3_EStop : DCI_STOP;   // Status of E-Stop 3
   MC_3_EStop_Status : BOOL := 1;   // General status of inputs
   MC_4_EStop : DCI_STOP;   // Status of E-Stop 4
   MC_4_EStop_Status : BOOL := 1;   // General status of inputs
   MC_5_EStop : DCI_STOP;   // Status of E-Stop 5
   MC_5_EStop_Status : BOOL := 1;   // General status of inputs
   MC_6_EStop : DCI_STOP;
   MC_6_EStop_Status : BOOL;
   MC_LigthCurtain_Status : BOOL;
   MEMORIA_DELTA_INICIO : BOOL := 1;   // Inicio de delta
   Memory : BOOL;
   Mesa_Kuka_Piston_1_Abierto : BOOL;   // Pistón Designado Para Posición de Pieza 1 Abierto
   Mesa_Kuka_Piston_1_Cerrado : BOOL;   // Pistón Designado Para Posición de Pieza 1 Cerrado
   MotionGroup_Almacen_2 : MOTION_GROUP;
   MSA_Mtr_Alm_2 : MOTION_INSTRUCTION;
   MSF_Mtr_Alm_1 : MOTION_INSTRUCTION;
   MSF_Mtr_Alm_2 : MOTION_INSTRUCTION;
   MSO_Mtr_Alm_1 : MOTION_INSTRUCTION;
   MSO_Mtr_Alm_2 : MOTION_INSTRUCTION;
   MSO_OnDly : TIMER;
   Mtr_Alm_1 : MOTION_INSTRUCTION;
   Mtr_Alm_1_Actual_pos : DINT;
   Mtr_Alm_1_Select_Pos : DINT := 1;
   Mtr_Alm_1_Speed : DINT := 20;
   Mtr_Alm_2 : MOTION_INSTRUCTION;
   Mtr_Alm_2_Speed : DINT := 50;
   New_count : COUNTER;
   ok : BOOL;
   ok_01 : Safety;
   ok_123 : Safety;
   ok_com : BOOL := 1; {access Read Only}   // tag de prueba de comunicacion
   Ons : INT := 5;
   Open_Griper_Fanuc : BOOL := 1;   // Señal De Griper Abierto Robot Fanuc
   Operation_Mode : BOOL := 1;   // Operation Mode for HMI (1) Manual (0) Automatico
   OSR_Alm_1 : BOOL;
   OSR_OB_Alm1 : BOOL;
   Paro_Emergencia_Almacen_1 : BOOL;   // Stopping signal of Torc Off Almacen 1
   Paro_Emergencia_Almacen_2 : BOOL;   // Stopping signal of Torc Off Almacen 2
   Permissive_Step0 : BOOL;
   Permissive_Step1 : BOOL;
   Permissive_Step10 : BOOL;
   Permissive_Step11 : BOOL;
   Permissive_Step12 : BOOL;
   Permissive_Step13 : BOOL;
   Permissive_Step14 : BOOL;
   Permissive_Step15 : BOOL;
   Permissive_Step16 : BOOL;
   Permissive_Step17 : BOOL;
   Permissive_Step18 : BOOL;
   Permissive_Step19 : BOOL;
   Permissive_Step2 : BOOL;
   Permissive_Step20 : BOOL;
   Permissive_Step21 : BOOL;
   Permissive_Step22 : BOOL;
   Permissive_Step23 : BOOL;
   Permissive_Step24 : BOOL;
   Permissive_Step25 : BOOL;
   Permissive_Step26 : BOOL;
   Permissive_Step27 : BOOL;
   Permissive_Step28 : BOOL;
   Permissive_Step29 : BOOL;
   Permissive_Step3 : BOOL;
   Permissive_Step30 : BOOL;
   Permissive_Step4 : BOOL;
   Permissive_Step5 : BOOL;
   Permissive_Step6 : BOOL;
   Permissive_Step7 : BOOL;
   Permissive_Step8 : BOOL;
   Permissive_Step9 : BOOL;
   PF_ClearFault_525_Conv_1 : BOOL;   // Clear Fault PowerFlex Conveyor 1
   PF_Jog_525_Conv_1 : BOOL;   // Miovimiento Jog PowerFlex Conveyor 1
   PF_On_525_Conv_1 : BOOL;   // Encender/Apagar PowerFlex Conveyor 1
   PickPosition : Position_Storage;
   PickPosition1 : Position_Storage;
   Pieza_Posicion_Prensa_CNC_1 : BOOL := 1;
   Pieza_Salida_Prensa_CNC_1 : BOOL := 1;
   Piston_CambioDir_Almacen_Conv_1 : BOOL;   // Cambiar Direccion de Pieza Lado Almacen Conveyor 1
   Piston_CambioDir_Almacen_Conv_2 : BOOL;   // Cambiar Direccion de Pieza Lado Almacen Conveyor 2
   Piston_CambioDir_CNC_Conv_1 : BOOL;   // Cambiar Dirección de Pieza Lado CNC Conveyor 1
   Piston_CambioDir_CNC_Conv_2 : BOOL;   // Cambiar Dirección de Pieza Lado CNC Conveyor 2
   Piston_Horizontal_Conv_1 : BOOL;   // Extender Pistón Horizontal del Conveyor 1
   Piston_Horizontal_Conv_2 : BOOL;   // Extender Pistón Horizontal del Conveyor 2
   PIT : BOOL;
   PLC_Com : DINT; {produced}
   Pos_4_Kinetix : BOOL;
   Pos_5_Kinetix : BOOL;
   Pos_6_Kinetix : BOOL;
   PosGrua1 : DINT;
   PosGrua2 : DINT := 20;
   PosicionAlmacen : DINT;
   PosMatrix : DINT[2,10] := ([0,1] := -23, [0,2] := 157, [0,3] := 337, [0,4] := 517, [0,5] := 697, [0,6] := 877, [0,8] := 325, [0,9] := 360, [1,1] := -23, [1,2] := 157, [1,3] := 337, [1,4] := 517, [1,5] := 697, [1,6] := 877);
   Prensa_Abierta_CNC_1 : BOOL := 1;   // Sensor de Prensa Abierta en CNC 1 Conveyor 1
   Prensa_Abierta_CNC_2 : BOOL := 1;   // Sensor de Prensa Abierta en CNC 2 Conveyor 2
   Prensa_Cerrada_CNC_1 : BOOL := 1;   // Sensor de Prensa Cerrada en CNC 1 Conveyor 1
   Prioridad_Pieza_1 : BOOL;
   Prioridad_Pieza_2 : BOOL;
   Prioridad_Pza_1 : DINT;
   Prioridad_Pza_2 : DINT;
   Produced_Signals_TEC_81_Conveyor_1 : DINT; {produced}
   Programa_CNC_1_Terminado : BOOL;
   Programa_CNC_2_Terminado : BOOL;
   Puerta_Abierta_CNC_1 : BOOL;   // Sensor de Puerta Abierta en CNC 1 Conveyor 1
   Puerta_Abierta_CNC_1_Sty : BOOL;
   Puerta_Abierta_CNC_2 : BOOL;   // Sensor de Puerta Abierta en CNC 2 Conveyor 2
   Puerta_Cerrada_CNC_1 : BOOL;   // Señal de Electroválvula para confirmar puerta cerrada en CNC 1
   Puerta_Cerrada_CNC_2 : BOOL;
   Pulse : TIMER;
   PV_ClearFaults : BOOL;
   PV_Cmd_Axis_2 : BOOL;
   PV_Hold : BOOL;
   PV_Hold_Alm1 : BOOL;
   PV_JogDwn : BOOL;
   PV_JogUp : BOOL;
   PV_ManPos : DINT := 380;
   PV_Mtr_Alm_1_Speed : DINT := 20;
   PV_Mtr_Alm_2_Speed : DINT := 50;
   PV_ServoOFF : BOOL;
   Pza_Lista_Conv1_To_CNC_1 : BOOL;   // Pieza en Espera de ser Tomada por Robot Fanuc para ser Llevada a CNC 1
   Pza_Lista_Conv2_To_CNC_2 : BOOL;   // Pieza en Espera de ser Tomada por Robot Fanuc para ser Llevada a CNC 2
   Reset_Almacen_1 : BOOL;
   Reset_Almacen_1_Sfty : BOOL;
   Reset_almacen_2 : BOOL;
   Reset_Almacen_2_Sfty : BOOL;
   Reset_Conveyor_1_Sfty : BOOL;
   Reset_Conveyor_2_Sfty : BOOL;
   reset_Kinetix : BOOL;
   Reset_PF525_Almacen_1 : DINT; {produced}
   Reset_PF525_Almacen_2 : DINT; {produced}
   Reset_Principal : BOOL;
   Reset_Principal_Sfty : BOOL;
   Reset_Salida_1 : BOOL;
   Reset_Salida_1_Sfty : BOOL;
   Retorno_Pieza_A_Conveyor_1 : BOOL;
   Retorno_Pieza_A_Conveyor_2 : BOOL;
   Retraer_Piston_1_Mesa_Kuka : BOOL;   // Retraer Pistón Esquina de Mesa Central
   Retraer_Piston_2_Mesa_Kuka : BOOL := 1;   // Retraer Pistón Centro de Mesa Central
   Robot_a : BOOL;
   Robot_Fuera_CNC_1_Prueba : BOOL;
   Robot_Fuera_CNC_2_Prueba : BOOL;
   Robot_Pieza_1_Kuka : BOOL;   // Robot Fanuc Deja Pieza Terminada de CNC 1 en Mesa de Robot Kuka
   Robot_Pieza_2_Kuka : BOOL;   // Robot Fanuc Deja Pieza Terminada de CNC 2 en Mesa de Robot Kuka
   Robot_Seq_Actual_Step : DINT;
   Robot_Seq_Perm_OnDly : TIMER[31];
   Robot_Step : DINT := 1;
        .1   // DECIDE QUE RUTINA EJECUTAR
        .20   // ROBOT COLOCA PIEZA EN CNC 2
        .21   // CIERRA PUERTA CNC 2
        .22   // INICIA CICLO CNC 2
        .23   // ROBOT TOMA PIEZA DE CNC 2 Y LA COLOCA EN MESA CENTRAL
        .24   // CIERRA GRIPPER DE MESA CENTRAL
        .25   // ROBOT TOMA PIEZA DE MESA CENTRAL Y LA REGRESA A TRANSPORTADOR 2
   Safety_FromTEC81 : Safety; {produced}
        .DINT.0   // Safety Close Loop OK
        .DINT.6   // Safety Torc Off Almacen 2
        .DINT.2   // Laser Scanner OK
        .DINT.5   // Operation Mode status (0) Automatic (1) Manual
        .DINT.1   // Interlock OK
        .DINT.7   // Safety Torc Off Almacen 1
        .DINT.4   // Mat OK
        .DINT.3   // Light Courtains OK
   Safety_Test_Bit : DINT;
   SafetyReset_almacen_1 : BOOL;   // Reset status Almacen 1
   SafetyReset_almacen_2 : BOOL;   // Reset status Almacen 2
   SafetyReset_Conveyor_1 : BOOL;
   SafetyReset_Conveyor_2 : BOOL;
   SafetyReset_Principal : BOOL;   // Reset status salida principal
   SafetyReset_Salida_1 : BOOL;   // Reset status Salida 1
   Sensor_Difuso_1_1_Conv_1 : BOOL;   // Sensor Lado A Almacen 1-1
   Sensor_Difuso_1_1_Conv_2 : BOOL;   // Sensor Difuso Presencia Lado A Almacen 1-1
   Sensor_Difuso_1_2_Conv_1 : BOOL;   // Sensor Lado A Almacen 1-2
   Sensor_Difuso_1_2_Conv_2 : BOOL;   // Sensor Difuso Presencia Lado A Almacén 1-2
   Sensor_Difuso_2_1_Conv_1 : BOOL;   // Sensor Lado B Almacen 2-1
   Sensor_Difuso_2_1_Conv_2 : BOOL;   // Sensor Difuso Presencia Lado B CNC 2-1
   Sensor_Difuso_2_2_Conv_1 : BOOL;   // Sensor Lado B Almacen 2-2
   Sensor_Difuso_2_2_Conv_2 : BOOL;   // Sensor Difuso Presencia Lado B CNC 2-2
   Sensor_Difuso_3_1_Conv_1 : BOOL;   // Sensor Lado A CNC 3-1
   Sensor_Difuso_3_1_Conv_2 : BOOL;   // Sensor Difuso Presencia Lado A CNC 3-1
   Sensor_Difuso_3_2_Conv_1 : BOOL;   // Sensor Lado A CNC 3-2
   Sensor_Difuso_3_2_Conv_2 : BOOL;   // Sensor Difuso Presencia Lado A CNC 3-2
   Sensor_Griper_Fanuc_Abierto : BOOL := 1;   // Sensor Indicador Griper en Robot Fanuc Abierto
   Sensor_Griper_Fanuc_Cerrado : BOOL;   // Sensor Indicador Griper en Robot Fanuc Cerrado
   Sensor_Inductivo_Alimentacion_Conv_1 : BOOL;   // Sensor Inductivo Alimentacion y Salida Almacen Conveyor 1
   Sensor_Inductivo_Almacen_Conv_1 : BOOL;   // Sensor Inductivo Lado A Final derecha Almacen
   Sensor_Inductivo_Almacen_Conv_2 : BOOL;   // Sensor Inductivo Lado A Almacén (Entrada)
   Sensor_Inductivo_CNC_2_Conv_1 : BOOL;   // Sensor Inductivo Lado B CNC
   Sensor_Inductivo_CNC_2_Conv_2 : BOOL;   // Sensor Inductivo Posición Lado A CNC
   Sensor_Inductivo_CNC_Conv_1 : BOOL;   // Sensor Inductivo Lado A CNC
   Sensor_Inductivo_CNC_Conv_2 : BOOL;   // Sensor Inductivo Posición Lado B CNC
   Sensor_Inductivo_Entrada_Conv_1 : BOOL;   // Sensor Inductivo Entrada Lado CNC (Adelante)
   Sensor_Inductivo_Entrada_Conv_2 : BOOL;   // Sensor Inductivo Lado B CNC (Entrada) Conveyor 2
   Sensor_Inductivo_Limit_Conv_2 : BOOL;   // Sensor Inductivo Limit Switch (Revisarl, Empate)
   Sensor_Inductivo_Marcadora : BOOL;   // Sensor Inductivo Presencia Zona Marcadora Laser
   Sensor_Inductivo_Salida_Conv_2 : BOOL;   // Sensor Inductivo a Salida/entrada Almacen
   Sensor_Inductivo_Vision_Conv_2 : BOOL;   // Sensor Presencia Zona de Marcadora Láser
   Sensor_Limit_Up_Conv_1 : BOOL;   // Limit Switch Arriba
   Sensor_Limit_Up_Conv_2 : BOOL;   // Limit Switch Arriba
   Sensor_PH_Ext_Conv_1 : BOOL;   // Sensor Pistón Horizontal Extendido
   Sensor_PH_Ret_Conv_1 : BOOL := 1;   // Sensor Pistón Horizontal Retraido
   Sensor_PistHor_Ext_Conv_2 : BOOL;   // Sensor Pistón Horizontal Extendido
   Sensor_PistHor_Ret_Conv_2 : BOOL;   // Sensor Pistón Horizontal Retraido
   Sensor_Piston_1_Ext_Mesa : BOOL;   // Sensor de Piston Extendido Esquina de la Mesa Central
   Sensor_Piston_1_Ret_Mesa : BOOL;   // Sensor de Pistón Retraido Esquina de la Mesa Central
   Sensor_Piston_2_Ext_Mesa : BOOL;   // Sensor de Pistón Extendido Centro de la Mesa Central
   Sensor_Piston_2_Ret_Mesa : BOOL;   // Sensor de Pistón Retraido Centro de la Mesa Central
   Sensor_Piston_Ext_Centro_Mesa_Prueba : BOOL;
   Sensor_Piston_Ext_Esquina_Mesa_Prueba : BOOL;
   Sensor_Piston_Ret_Centro_Mesa_Prueba : BOOL;
   Sensor_Piston_Ret_Esquina_Mesa_Prueba : BOOL;
   Sensor_Prensa_Abierta_CNC_1 : BOOL;
   Sensor_Prensa_Abierta_CNC_2 : BOOL;
   Sensor_Prensa_Cerrada_CNC_1 : BOOL := 1;
   Sensor_Prensa_Cerrada_CNC_2 : BOOL;
   Sensor_Tope_CNC_Conv_1 : BOOL;   // Sensor Pistón Tope CNC
   Sensor_Tope_CNC_Conv_2 : BOOL;   // Sensor Tope Pistón CNC
   Sensor_Tope_Marcadora_Conv_1 : BOOL;   // Sensor Pistón Tope Marcadora Láser
   Sensor_Tope_Marcadora_Conv_2 : BOOL;   // Sensor Pistón Tope Marcadora Láser
   Sensor_Tope_PH_Conv_1 : BOOL;   // Sensor Tope Pistón Horizontal
   Sensor_Tope_PH_Conv_2 : BOOL;   // Sensor Tope Pistón Horizontal (Salida de Conveyor 2)
   Sensor_Tope_Vision_Conv_1 : BOOL;   // Sensor Pistón Tope Cámara de Visión
   Sensor_Tope_Vision_Conv_2 : BOOL;   // Sensor Pistón Tope Cámara de Visión
   Sequence_Salida_Conv_1 : BOOL;   // Secuencia de Salida de Producto Maquinado Retorno a Almacén
   Sequence_Start_Conv_1 : BOOL;   // Inicia Secuenca Automática con Pieza Conveyor 1
   Servo_Alm_1_On : BOOL;
   Servo_Alm_1_Reset : BOOL;
   Servo_Alm_1_Start : BOOL;
   servo_start : MOTION_INSTRUCTION;
   servo_start_01 : MOTION_INSTRUCTION;
   Sevo_home : BOOL;
   Sevo_Stop : MOTION_INSTRUCTION;
   Signal_Fanuc_Tomar_Pieza_Conv_1 : BOOL;   // Señal para Tomar pieza desde el Conveyor 1 Hacia CNC
   Slector_Automatico_Conv_1 : BOOL := 1;   // Bit Selector Automático ON
   Start_Kinetix_Alm_1 : DINT;
   Start_Kinetix_Alm_2 : DINT := 1;
   Start_Robot_Seq : BOOL;
   Start_Servo : BOOL := 1;
   Step0 : BOOL;   // StandBy
   Step1 : BOOL;   // Y Safe Position
   Step10 : BOOL;
   Step11 : BOOL;
   step12 : BOOL;
   step13 : BOOL;
   Step14 : BOOL;
   Step15 : DINT;
   Step16 : DINT;
   Step17 : BOOL;
   Step18 : BOOL;
   Step19 : BOOL;
   Step2 : BOOL;   // Opening Gripper
   Step20 : BOOL;
   Step21 : BOOL;
   Step22 : BOOL;
   Step23 : BOOL;
   Step24 : BOOL;
   Step25 : BOOL;
   Step26 : BOOL;
   Step27 : BOOL;
   Step28 : BOOL;
   Step29 : BOOL;
   Step3 : BOOL;   // Stacker Safe Position
   Step30 : BOOL;
   Step4 : BOOL;   // Move Z Safe Position
   Step5 : BOOL;   // Storage SafePosition
   Step6 : BOOL;   // Y to Y Safe to Pick
   Step7 : BOOL;   // Move X To X Pick
   Step8 : BOOL;
   step9 : BOOL;
   Step_00_Robot : BOOL;
   Step_11_Robot : BOOL;
   Step_12_Robot : BOOL;
   Step_13_Robot : BOOL;
   Step_14_Robot : BOOL;
   Step_15_Robot : BOOL;
   Step_16_Robot : BOOL;
   Step_17_Robot : BOOL;
   Step_18_Robot : BOOL;
   Step_19_Robot : BOOL;
   Step_200_Pieza : BOOL := 1;
   Step_200A_Pieza : BOOL;
   Step_201_Pieza : BOOL;
   Step_201A_Pieza : BOOL;
   Step_202_Pieza : BOOL;
   Step_203_Pieza : BOOL;
   Step_204_Pieza : BOOL;
   Step_205_Pieza : BOOL;
   Step_206_Pieza : BOOL;
   Step_207_Pieza : BOOL;
   Step_208_Pieza : BOOL;
   Step_209_Pieza : BOOL;
   Step_209A_Pieza : BOOL;
   Step_210_Pieza : BOOL;
   Step_211_Pieza : BOOL;
   Step_212_Pieza : BOOL;
   Step_213_Pieza : BOOL;
   Step_214_Pieza : BOOL;
   Step_215_Pieza : BOOL;
   Step_216_Pieza : BOOL;
   Step_217_Pieza : BOOL;
   Step_217A_Pieza : BOOL;
   Step_218_Pieza : BOOL;
   Step_219_Pieza : BOOL;
   Step_21_Robot : BOOL;
   Step_220_Pieza : BOOL;
   Step_221_Pieza : BOOL;
   Step_221A_Pieza : BOOL;
   Step_222_Pieza : BOOL;
   Step_223_Pieza : BOOL;
   Step_224_Pieza : BOOL;
   Step_225_Pieza : BOOL;
   Step_226_Pieza : BOOL;
   Step_227_Pieza : BOOL;
   Step_228_Pieza : BOOL;
   Step_229_Pieza : BOOL;
   Step_22_Robot : BOOL;
   Step_230_Pieza : BOOL;
   Step_231_Pieza : BOOL;
   Step_232_Pieza : BOOL;
   Step_233_Pieza : BOOL;
   Step_234_Pieza : BOOL;
   Step_235_Pieza : BOOL;
   Step_236_Pieza : BOOL;
   Step_237_Pieza : BOOL;
   Step_238_Pieza : BOOL;
   Step_239_Pieza : BOOL;
   Step_23_Robot : BOOL;
   Step_240_Pieza : BOOL;
   Step_241_Pieza : BOOL;
   Step_24_Robot : BOOL;
   Step_25_Robot : BOOL;
   Step_26_Robot : BOOL;
   Step_300_Pieza_2 : BOOL := 1;
   Step_301_Pieza_2 : BOOL;
   Step_302_Pieza_2 : BOOL;
   Step_303_Pieza_2 : BOOL;
   Step_304_Pieza_2 : BOOL;
   Step_304A_Pieza_2 : BOOL;
   Step_304B_Pieza_2 : BOOL;
   Step_305_Pieza_2 : BOOL;
   Step_306_Pieza_2 : BOOL;
   Step_307_Pieza_2 : BOOL;
   Step_308_Pieza_2 : BOOL;
   Step_309_Pieza_2 : BOOL;
   Step_310_Pieza_2 : BOOL;
   Step_311_Pieza_2 : BOOL;
   Step_312_Pieza_2 : BOOL;
   Step_313_Pieza_2 : BOOL;
   Step_314_Pieza_2 : BOOL;
   Step_315_Pieza_2 : BOOL;
   Step_316_Pieza_2 : BOOL;
   Step_317_Pieza_2 : BOOL;
   Step_318_Pieza_2 : BOOL;
   Step_319_Pieza_2 : BOOL;
   Step_31_Robot : BOOL;
   Step_320_Pieza_2 : BOOL;
   Step_320A_Pieza_2 : BOOL;
   Step_321_Pieza_2 : BOOL;
   Step_322_Pieza_2 : BOOL;
   Step_323_Pieza_2 : BOOL;
   Step_324_Pieza_2 : BOOL;
   Step_325_Pieza_2 : BOOL;
   Step_326_Pieza_2 : BOOL;
   Step_327_Pieza_2 : BOOL;
   Step_328_Pieza_2 : BOOL;
   Step_329_Pieza_2 : BOOL;
   Step_32_Robot : BOOL;
   Step_330_Pieza_2 : BOOL;
   Step_331_Pieza_2 : BOOL;
   Step_332_Pieza_2 : BOOL;
   Step_333_Pieza_2 : BOOL;
   Step_334_Pieza_2 : BOOL;
   Step_335_Pieza_2 : BOOL;
   Step_336_Pieza_2 : BOOL;
   Step_337_Pieza_2 : BOOL;
   Step_338_Pieza_2 : BOOL;
   Step_339_Pieza_2 : BOOL;
   Step_33_Robot : BOOL;
   Step_340_Pieza_2 : BOOL;
   Step_341_Pieza_2 : BOOL;
   Step_342_Pieza_2 : BOOL;
   Step_343_Pieza_2 : BOOL;
   Step_344_Pieza_2 : BOOL;
   Step_345_Pieza_2 : BOOL;
   Step_346_Pieza_2 : BOOL;
   Step_347_Pieza_2 : BOOL;
   Step_348_Pieza_2 : BOOL;
   Step_349_Pieza_2 : BOOL;
   Step_34_Robot : BOOL;
   Step_350_Pieza_2 : BOOL;
   Step_351_Pieza_2 : BOOL;
   Step_352_Pieza_2 : BOOL;
   Step_353_Pieza_2 : BOOL;
   Step_354_Pieza_2 : BOOL;
   Step_355_Pieza_2 : BOOL;
   Step_356_Pieza_2 : BOOL;
   Step_357_Pieza_2 : BOOL;
   Step_358_Pieza_2 : BOOL;
   Step_359_Pieza_2 : BOOL;
   Step_360_Pieza_2 : BOOL;
   Step_41_Robot : BOOL;
   Step_42_Robot : BOOL;
   Step_43_Robot : BOOL;
   Step_44_Robot : BOOL;
   Step_45_Robot : BOOL;
   Step_46_Robot : BOOL;
   Step_47_Robot : BOOL;
   Step_48_Robot : BOOL;
   Step_51_Robot : BOOL;
   Step_52_Robot : BOOL;
   Step_53_Robot : BOOL;
   Step_54_Robot : BOOL;
   Step_55_Robot : BOOL;
   Step_56_Robot : BOOL;
   Step_57_Robot : BOOL;
   Step_58_Robot : BOOL;
   Step_Pieza : DINT := 200;
   Step_Pieza_2 : DINT := 300;
   Step_Robot : DINT;
   Stop_Servo : BOOL;
   Storage_1 : BOOL;
   Storage_1_Y_ActualPosition : REAL; {produced}
   Storage_2 : BOOL;
   Storage_2_Y_ActualPosition : REAL; {produced}
   Storage_3 : BOOL;
   Storage_4 : BOOL;
   Storage_5 : BOOL;
   Storage_6 : BOOL;
   Sts_Auto : BOOL := 1;
   T_Espera_Pza_1 : TIMER;
   T_Espera_Pza_2 : TIMER;
   T_Fanuc_A_Conv_1 : TIMER;
   T_Fanuc_A_Conv_2 : TIMER;
   T_Permisive_Step_00_Robot : TIMER;
   T_Permisive_Step_200 : TIMER;
   T_Permisive_Step_200A : TIMER;
   T_Permisive_Step_201 : TIMER;
   T_Permisive_Step_201A : TIMER;
   T_Permisive_Step_202 : TIMER;
   T_Permisive_Step_203 : TIMER;
   T_Permisive_Step_204 : TIMER;
   T_Permisive_Step_205 : TIMER;
   T_Permisive_Step_206 : TIMER;
   T_Permisive_Step_207 : TIMER;
   T_Permisive_Step_208 : TIMER;
   T_Permisive_Step_209 : TIMER;
   T_Permisive_Step_209A : TIMER;
   T_Permisive_Step_210 : TIMER;
   T_Permisive_Step_211 : TIMER;
   T_Permisive_Step_212 : TIMER;
   T_Permisive_Step_213 : TIMER;
   T_Permisive_Step_214 : TIMER;
   T_Permisive_Step_215 : TIMER;
   T_Permisive_Step_216 : TIMER;
   T_Permisive_Step_217 : TIMER;
   T_Permisive_Step_217A : TIMER;
   T_Permisive_Step_218 : TIMER;
   T_Permisive_Step_219 : TIMER;
   T_Permisive_Step_220 : TIMER;
   T_Permisive_Step_221 : TIMER;
   T_Permisive_Step_221A : TIMER;
   T_Permisive_Step_222 : TIMER;
   T_Permisive_Step_223 : TIMER;
   T_Permisive_Step_224 : TIMER;
   T_Permisive_Step_225 : TIMER;
   T_Permisive_Step_226 : TIMER;
   T_Permisive_Step_227 : TIMER;
   T_Permisive_Step_228 : TIMER;
   T_Permisive_Step_229 : TIMER;
   T_Permisive_Step_230 : TIMER;
   T_Permisive_Step_231 : TIMER;
   T_Permisive_Step_232 : TIMER;
   T_Permisive_Step_233 : TIMER;
   T_Permisive_Step_234 : TIMER;
   T_Permisive_Step_235 : TIMER;
   T_Permisive_Step_236 : TIMER;
   T_Permisive_Step_237 : TIMER;
   T_Permisive_Step_238 : TIMER;
   T_Permisive_Step_239 : TIMER;
   T_Permisive_Step_240 : TIMER;
   T_Permisive_Step_241 : TIMER;
   T_Permisive_Step_300 : TIMER;
   T_Permisive_Step_301 : TIMER;
   T_Permisive_Step_302 : TIMER;
   T_Permisive_Step_303 : TIMER;
   T_Permisive_Step_304 : TIMER;
   T_Permisive_Step_304A : TIMER;
   T_Permisive_Step_304B : TIMER;
   T_Permisive_Step_305 : TIMER;
   T_Permisive_Step_306 : TIMER;
   T_Permisive_Step_307 : TIMER;
   T_Permisive_Step_308 : TIMER;
   T_Permisive_Step_309 : TIMER;
   T_Permisive_Step_310 : TIMER;
   T_Permisive_Step_311 : TIMER;
   T_Permisive_Step_312 : TIMER;
   T_Permisive_Step_313 : TIMER;
   T_Permisive_Step_314 : TIMER;
   T_Permisive_Step_315 : TIMER;
   T_Permisive_Step_316 : TIMER;
   T_Permisive_Step_317 : TIMER;
   T_Permisive_Step_318 : TIMER;
   T_Permisive_Step_319 : TIMER;
   T_Permisive_Step_320 : TIMER;
   T_Permisive_Step_320A : TIMER;
   T_Permisive_Step_321 : TIMER;
   T_Permisive_Step_322 : TIMER;
   T_Permisive_Step_323 : TIMER;
   T_Permisive_Step_324 : TIMER;
   T_Permisive_Step_325 : TIMER;
   T_Permisive_Step_326 : TIMER;
   T_Permisive_Step_327 : TIMER;
   T_Permisive_Step_328 : TIMER;
   T_Permisive_Step_329 : TIMER;
   T_Permisive_Step_330 : TIMER;
   T_Permisive_Step_331 : TIMER;
   T_Permisive_Step_332 : TIMER;
   T_Permisive_Step_333 : TIMER;
   T_Permisive_Step_334 : TIMER;
   T_Permisive_Step_335 : TIMER;
   T_Permisive_Step_336 : TIMER;
   T_Permisive_Step_337 : TIMER;
   T_Permisive_Step_338 : TIMER;
   T_Permisive_Step_339 : TIMER;
   T_Permisive_Step_340 : TIMER;
   T_Permisive_Step_341 : TIMER;
   T_Permisive_Step_342 : TIMER;
   T_Permisive_Step_343 : TIMER;
   T_Permisive_Step_344 : TIMER;
   T_Permisive_Step_345 : TIMER;
   T_Permisive_Step_346 : TIMER;
   T_Permisive_Step_347 : TIMER;
   T_Permisive_Step_348 : TIMER;
   T_Permisive_Step_349 : TIMER;
   T_Permisive_Step_350 : TIMER;
   T_Permisive_Step_351 : TIMER;
   T_Permisive_Step_352 : TIMER;
   T_Permisive_Step_353 : TIMER;
   T_Permisive_Step_354 : TIMER;
   T_Permisive_Step_355 : TIMER;
   T_Permisive_Step_356 : TIMER;
   T_Permisive_Step_357 : TIMER;
   T_Permisive_Step_358 : TIMER;
   T_Permisive_Step_359 : TIMER;
   T_Permisive_Step_360 : TIMER;
   T_Permissive_Step0 : TIMER;
   T_Permissive_Step1 : TIMER;
   T_Permissive_Step10 : TIMER;
   T_Permissive_Step11 : TIMER;
   T_Permissive_Step12 : TIMER;
   T_Permissive_Step13 : TIMER;
   T_Permissive_Step14 : TIMER;
   T_Permissive_Step15 : TIMER;
   T_Permissive_Step16 : TIMER;
   T_Permissive_Step17 : TIMER;
   T_Permissive_Step18 : TIMER;
   T_Permissive_Step19 : TIMER;
   T_Permissive_Step2 : TIMER;
   T_Permissive_Step20 : TIMER;
   T_Permissive_Step21 : TIMER;
   T_Permissive_Step22 : TIMER;
   T_Permissive_Step23 : TIMER;
   T_Permissive_Step24 : TIMER;
   T_Permissive_Step25 : TIMER;
   T_Permissive_Step26 : TIMER;
   T_Permissive_Step27 : TIMER;
   T_Permissive_Step28 : TIMER;
   T_Permissive_Step29 : TIMER;
   T_Permissive_Step3 : TIMER;
   T_Permissive_Step30 : TIMER;
   T_Permissive_Step4 : TIMER;
   T_Permissive_Step5 : TIMER;
   T_Permissive_Step6 : TIMER;
   T_Permissive_Step7 : TIMER;
   T_Permissive_Step8 : TIMER;
   T_Permissive_Step9 : TIMER;
   Tec81_to_Wh2 : DINT; {produced}
   Test : BOOL;
   Test2 : BOOL;
   Test_Ali : BOOL;
   Test_Bit : DINT := 4132;
   Test_Bit_CNC_1 : BOOL := 1;
   Test_Bit_CNC_1_1 : BOOL := 1;
   Test_Caleb : BOOL;
   test_com : BOOL;   // bit e comunicacion
   Test_com_PLC : Safety;
   Test_Home : BOOL := 1;
   TEst_Leaa_Sfty : DINT := 3;
   TestHome : BOOL;
   To_Pos_Alm_1 : DINT := 64;
   To_Pos_Alm_2 : DINT := 128;
   To_Robot : ToRobot;
        .DI61   // CERRADO
        .DI60   // ABIERTO
        .DI25   // F
   TOF_STO_KinetixStorage2 : TIMER;
   tomas : BOOL;
   Tope_CNC_Conv_1 : BOOL;   // Tope Pistón CNC (Freno 5) Conveyor 1
   Tope_CNC_Conv_2 : BOOL;   // Tope Pistón CNC (Freno 5) Conveyor 2
   Tope_Marcadora_Conv_1 : BOOL;   // Tope Pistón Marcadora Láser (Freno 6) Conveyor 1
   Tope_Marcadora_Conv_2 : BOOL;   // Tope Pistón Marcadora Láser (Freno 6) Conveyor 2
   Tope_Salida_PH_Conv_1 : BOOL;   // Tope Pistón Salida de Producto (Freno 8) Conveyor 1
   Tope_Salida_PH_Conv_2 : BOOL;   // Tope Pistón Salida de Producto (Freno 8) Conveyor 2
   Tope_Vision_Conv_1 : BOOL;   // Tope Pistón Cáma de Visión Conveyor 1
   Tope_Vision_Conv_2 : BOOL;   // Tope Pistón Cámara de Visión Conveyor 2
   TT : BOOL;
   VentosaEnPosicion_Mesa : BOOL;   // Sensor de posición de Ventosa en Mesa Central
END_VAR

PROGRAM _05_Mesa_Central   (* main routine _01_Main *)

ROUTINE _01_Main   (* ladder *)
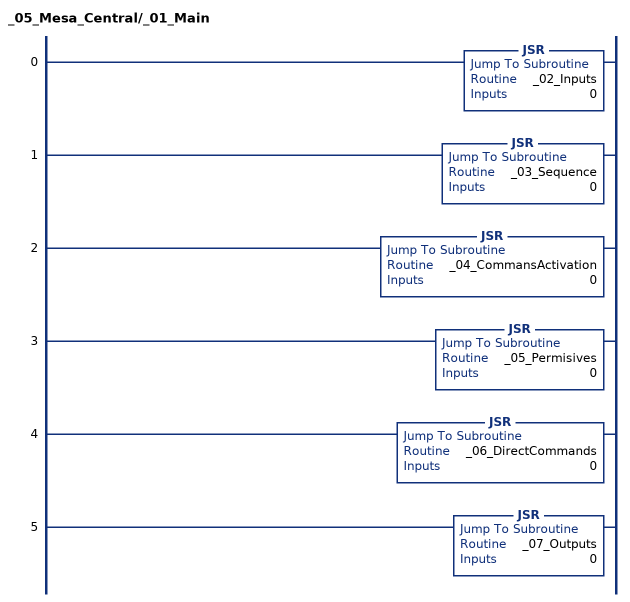
   0: JSR(_02_Inputs,0);
   1: JSR(_03_Sequence,0);
   2: JSR(_04_CommansActivation,0);
   3: JSR(_05_Permisives,0);
   4: JSR(_06_DirectCommands,0);
   5: JSR(_07_Outputs,0);
END_ROUTINE

ROUTINE _02_Inputs   (* ladder *)
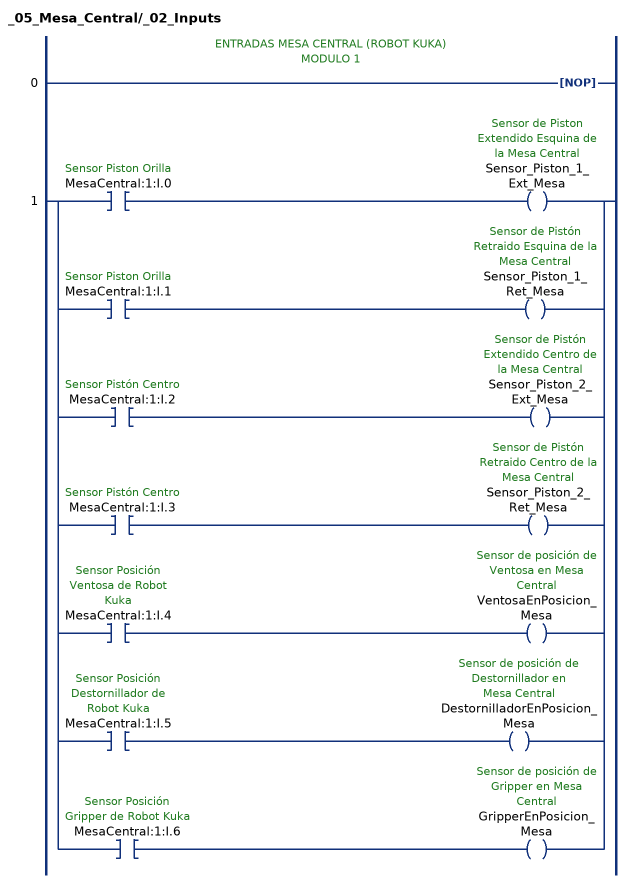
   // ENTRADAS MESA CENTRAL (ROBOT KUKA)
   // MODULO 1
   0: NOP();
   1: [XIC(MesaCentral:1:I.0) OTE(Sensor_Piston_1_Ext_Mesa) ,XIC(MesaCentral:1:I.1) OTE(Sensor_Piston_1_Ret_Mesa) ,XIC(MesaCentral:1:I.2) OTE(Sensor_Piston_2_Ext_Mesa) ,XIC(MesaCentral:1:I.3) OTE(Sensor_Piston_2_Ret_Mesa) ,XIC(MesaCentral:1:I.4) OTE(VentosaEnPosicion_Mesa) ,XIC(MesaCentral:1:I.5) OTE(DestornilladorEnPosicion_Mesa) ,XIC(MesaCentral:1:I.6) OTE(GripperEnPosicion_Mesa) ];
END_ROUTINE

ROUTINE _03_Sequence   (* ladder *)
END_ROUTINE

ROUTINE _04_CommansActivation   (* ladder *)
END_ROUTINE

ROUTINE _05_Permisives   (* ladder *)
END_ROUTINE

ROUTINE _06_DirectCommands   (* ladder *)
END_ROUTINE

ROUTINE _07_Outputs   (* ladder *)
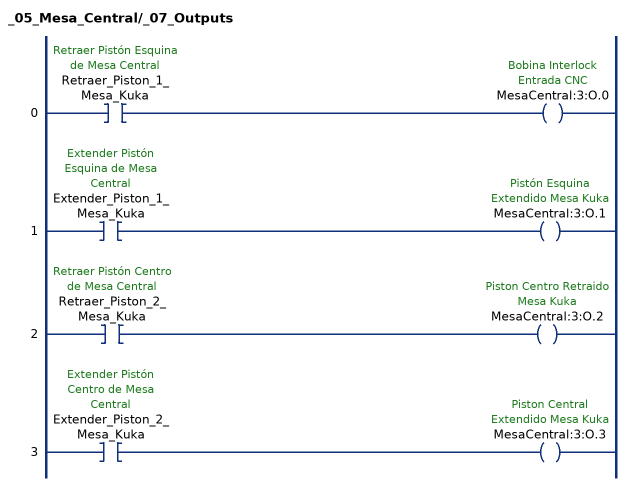
   0: XIC(Retraer_Piston_1_Mesa_Kuka)OTE(MesaCentral:3:O.0);
   1: XIC(Extender_Piston_1_Mesa_Kuka)OTE(MesaCentral:3:O.1);
   2: XIC(Retraer_Piston_2_Mesa_Kuka)OTE(MesaCentral:3:O.2);
   3: XIC(Extender_Piston_2_Mesa_Kuka)OTE(MesaCentral:3:O.3);
END_ROUTINE

ROUTINE test   (* sequential function chart *)
END_ROUTINE

ROUTINE test1   (* ladder *)
END_ROUTINE
END_PROGRAM

PROGRAM _Almacen_1   (* main routine _01_Main_Alm_11 *)
VAR
   B_Reset_Posicion_kinetix_0 : DINT := 319;
   Ctrl_Kinetix_A1 : DINT;
   Done_Kinetx_0 : DINT;
   home_step_1 : BOOL;
   Kinetix_Pos_Alm_0 : DINT;
   ok_com_1 : BOOL;
   reset_Kinetix_1 : BOOL;
END_VAR

ROUTINE _01_Main_Alm_11   (* ladder *)
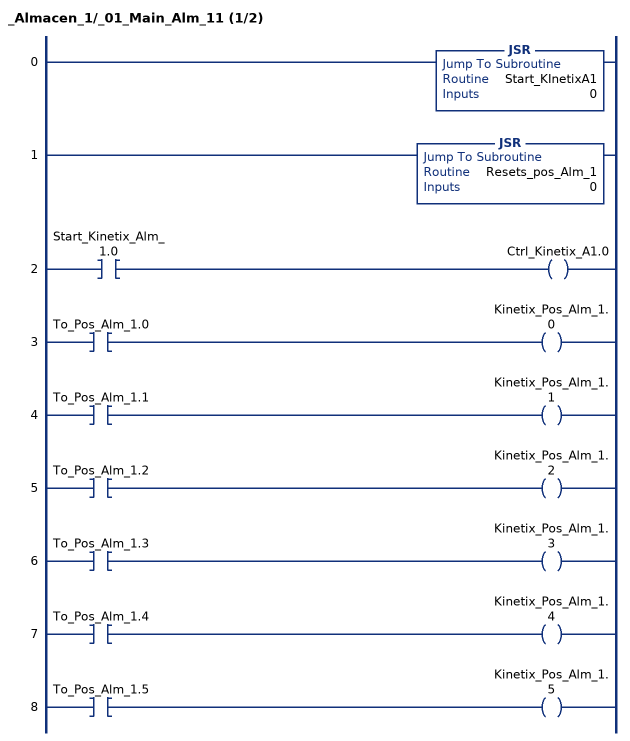
   0: JSR(Start_KInetixA1,0);
   1: JSR(Resets_pos_Alm_1,0);
   2: XIC(Start_Kinetix_Alm_1.0)OTE(Ctrl_Kinetix_A1.0);
   3: XIC(To_Pos_Alm_1.0)OTE(Kinetix_Pos_Alm_1.0);
   4: XIC(To_Pos_Alm_1.1)OTE(Kinetix_Pos_Alm_1.1);
   5: XIC(To_Pos_Alm_1.2)OTE(Kinetix_Pos_Alm_1.2);
   6: XIC(To_Pos_Alm_1.3)OTE(Kinetix_Pos_Alm_1.3);
   7: XIC(To_Pos_Alm_1.4)OTE(Kinetix_Pos_Alm_1.4);
   8: XIC(To_Pos_Alm_1.5)OTE(Kinetix_Pos_Alm_1.5);
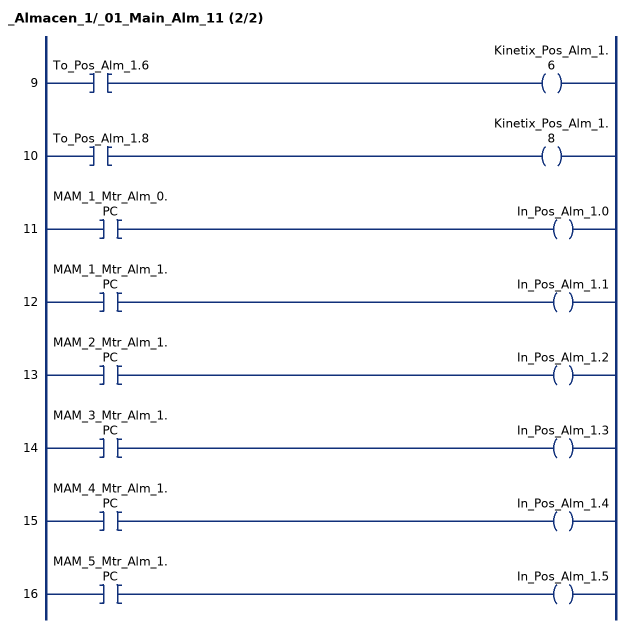
   9: XIC(To_Pos_Alm_1.6)OTE(Kinetix_Pos_Alm_1.6);
   10: XIC(To_Pos_Alm_1.8)OTE(Kinetix_Pos_Alm_1.8);
   11: XIC(MAM_1_Mtr_Alm_0.PC)OTE(In_Pos_Alm_1.0);
   12: XIC(MAM_1_Mtr_Alm_1.PC)OTE(In_Pos_Alm_1.1);
   13: XIC(MAM_2_Mtr_Alm_1.PC)OTE(In_Pos_Alm_1.2);
   14: XIC(MAM_3_Mtr_Alm_1.PC)OTE(In_Pos_Alm_1.3);
   15: XIC(MAM_4_Mtr_Alm_1.PC)OTE(In_Pos_Alm_1.4);
   16: XIC(MAM_5_Mtr_Alm_1.PC)OTE(In_Pos_Alm_1.5);
END_ROUTINE

ROUTINE Resets_pos_Alm_1   (* ladder *)
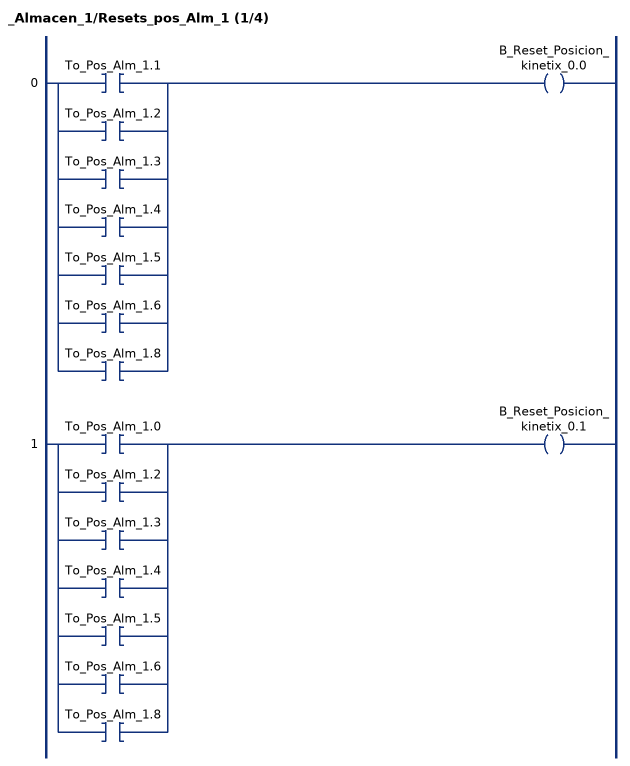
   0: [XIC(To_Pos_Alm_1.1) ,XIC(To_Pos_Alm_1.2) ,XIC(To_Pos_Alm_1.3) ,XIC(To_Pos_Alm_1.4) ,XIC(To_Pos_Alm_1.5) ,XIC(To_Pos_Alm_1.6) ,XIC(To_Pos_Alm_1.8) ]OTE(B_Reset_Posicion_kinetix_0.0);
   1: [XIC(To_Pos_Alm_1.0) ,XIC(To_Pos_Alm_1.2) ,XIC(To_Pos_Alm_1.3) ,XIC(To_Pos_Alm_1.4) ,XIC(To_Pos_Alm_1.5) ,XIC(To_Pos_Alm_1.6) ,XIC(To_Pos_Alm_1.8) ]OTE(B_Reset_Posicion_kinetix_0.1);
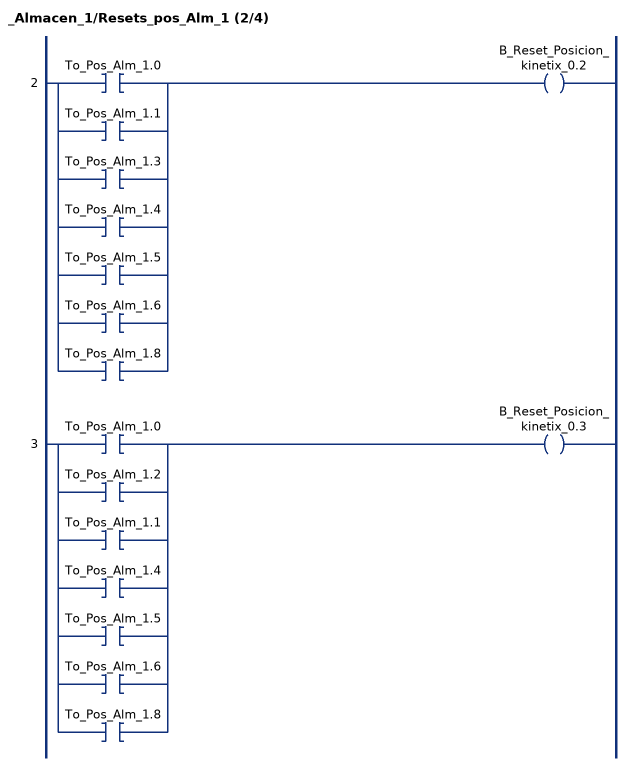
   2: [XIC(To_Pos_Alm_1.0) ,XIC(To_Pos_Alm_1.1) ,XIC(To_Pos_Alm_1.3) ,XIC(To_Pos_Alm_1.4) ,XIC(To_Pos_Alm_1.5) ,XIC(To_Pos_Alm_1.6) ,XIC(To_Pos_Alm_1.8) ]OTE(B_Reset_Posicion_kinetix_0.2);
   3: [XIC(To_Pos_Alm_1.0) ,XIC(To_Pos_Alm_1.2) ,XIC(To_Pos_Alm_1.1) ,XIC(To_Pos_Alm_1.4) ,XIC(To_Pos_Alm_1.5) ,XIC(To_Pos_Alm_1.6) ,XIC(To_Pos_Alm_1.8) ]OTE(B_Reset_Posicion_kinetix_0.3);
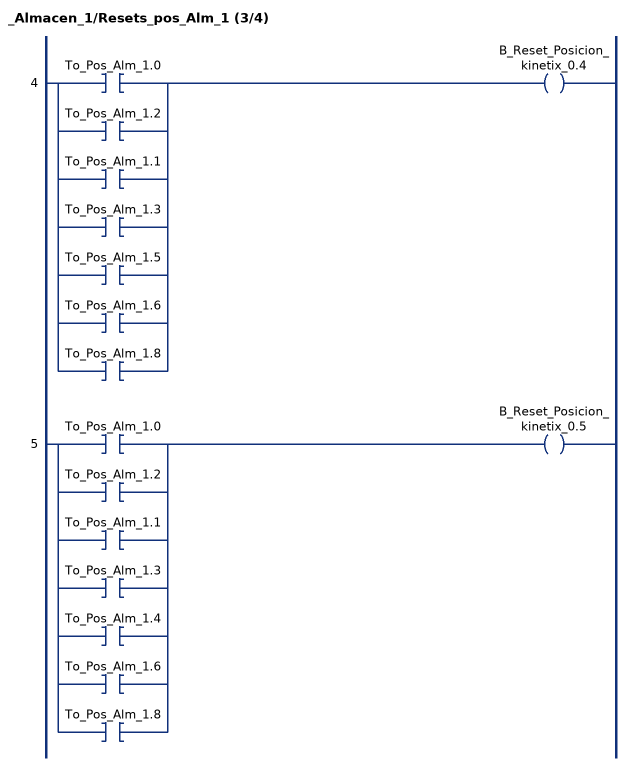
   4: [XIC(To_Pos_Alm_1.0) ,XIC(To_Pos_Alm_1.2) ,XIC(To_Pos_Alm_1.1) ,XIC(To_Pos_Alm_1.3) ,XIC(To_Pos_Alm_1.5) ,XIC(To_Pos_Alm_1.6) ,XIC(To_Pos_Alm_1.8) ]OTE(B_Reset_Posicion_kinetix_0.4);
   5: [XIC(To_Pos_Alm_1.0) ,XIC(To_Pos_Alm_1.2) ,XIC(To_Pos_Alm_1.1) ,XIC(To_Pos_Alm_1.3) ,XIC(To_Pos_Alm_1.4) ,XIC(To_Pos_Alm_1.6) ,XIC(To_Pos_Alm_1.8) ]OTE(B_Reset_Posicion_kinetix_0.5);
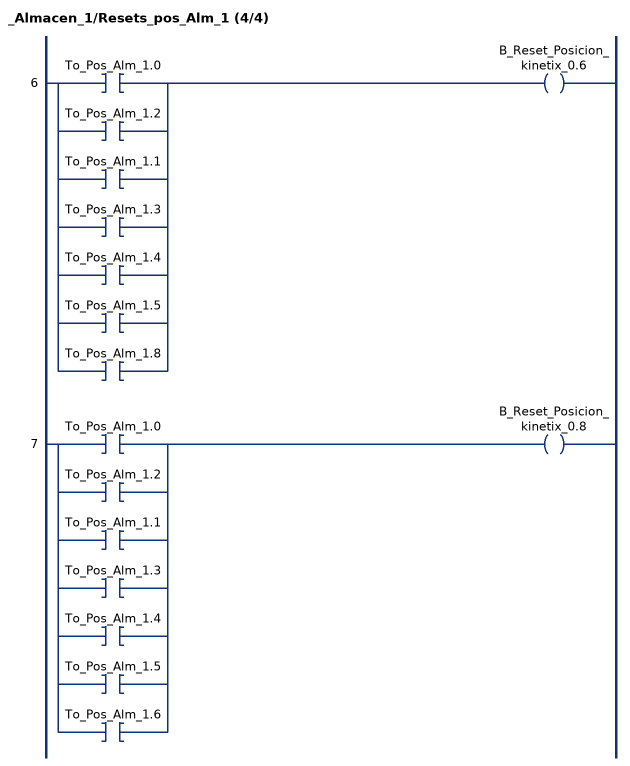
   6: [XIC(To_Pos_Alm_1.0) ,XIC(To_Pos_Alm_1.2) ,XIC(To_Pos_Alm_1.1) ,XIC(To_Pos_Alm_1.3) ,XIC(To_Pos_Alm_1.4) ,XIC(To_Pos_Alm_1.5) ,XIC(To_Pos_Alm_1.8) ]OTE(B_Reset_Posicion_kinetix_0.6);
   7: [XIC(To_Pos_Alm_1.0) ,XIC(To_Pos_Alm_1.2) ,XIC(To_Pos_Alm_1.1) ,XIC(To_Pos_Alm_1.3) ,XIC(To_Pos_Alm_1.4) ,XIC(To_Pos_Alm_1.5) ,XIC(To_Pos_Alm_1.6) ]OTE(B_Reset_Posicion_kinetix_0.8);
END_ROUTINE
